(* IEC 61131-3 sources: teller/JD_Teller_LC2_V11/Class/Box_Editer, 1 file *)

(* ---- Box_Editer.st ---- *)
(*!
<Class
	Name               = "Box_Editer"
	Revision           = "1.7"
	RealtimeTask       = "false"
	CyclicTask         = "false"
	BackgroundTask     = "false"
	Sigmatek           = "false"
	OSInterface        = "false"
	HighPriority       = "false"
	Automatic          = "false"
	UpdateMode         = "Prescan"
	SharedCommandTable = "true"
	Objectsize         = "(750,1860)">
	<Channels>
		<Server Name="ClassSvr" Visualized="false" Initialize="false" WriteProtected="true" Retentive="false"/>
		<Server Name="Parameter_Ok" Visualized="true" Initialize="false" WriteProtected="true" Retentive="false" Comment="Visu&#13;&#10;&#13;&#10;Als een doos berekend wordt dan wordt &#13;&#10;er gecontroleerd of de parameters kloppen&#13;&#10;&#13;&#10;Bij&#13;&#10;0: Fout&#13;&#10;1: Goed&#13;&#10;&#13;&#10;De servers T_Status, en verder geven de foute waarden per parameter aan&#13;&#10;"/>
		<Server Name="Presets_MinMax" Visualized="true" Initialize="false" WriteProtected="false" Retentive="false"/>
		<Server Name="ResetValues" Visualized="true" Initialize="false" WriteProtected="false" Retentive="false"/>
		<Server Name="s_BoxMogelijkopMachine" Visualized="true" Initialize="false" WriteProtected="false" Retentive="false" Comment="Is deze doos te draaien op de machine?&#13;&#10;&#13;&#10;0: nee&#13;&#10;1: ja&#13;&#10;"/>
		<Server Name="s_BoxType" Visualized="true" Initialize="false" WriteProtected="false" Retentive="SRam"/>
		<Server Name="s_Calc_Box" Visualized="true" Initialize="false" WriteProtected="false" Retentive="false"/>
		<Server Name="s_Doosnaam" Visualized="true" Initialize="false" WriteProtected="true" Retentive="false"/>
		<Server Name="s_MaxLength" Visualized="true" Initialize="false" WriteProtected="false" Retentive="false"/>
		<Server Name="s_MaxWidth" Visualized="true" Initialize="false" WriteProtected="false" Retentive="false"/>
		<Server Name="s_Offset" Visualized="true" Initialize="false" WriteProtected="false" Retentive="false"/>
		<Server Name="s_Offset_Max" Visualized="true" Initialize="false" WriteProtected="false" Retentive="false"/>
		<Server Name="s_Offset_Min" Visualized="true" Initialize="false" WriteProtected="false" Retentive="false"/>
		<Server Name="s_Refresh_Values" Visualized="false" Initialize="false" WriteProtected="false" Retentive="false"/>
		<Server Name="s_T" Visualized="true" Initialize="false" WriteProtected="false" Retentive="false"/>
		<Server Name="s_T_Max" Visualized="true" Initialize="false" WriteProtected="false" Retentive="false"/>
		<Server Name="s_T_Min" Visualized="true" Initialize="false" WriteProtected="false" Retentive="false"/>
		<Server Name="s_U" Visualized="true" Initialize="false" WriteProtected="false" Retentive="false"/>
		<Server Name="s_U_Max" Visualized="true" Initialize="false" WriteProtected="false" Retentive="false"/>
		<Server Name="s_U_Min" Visualized="true" Initialize="false" WriteProtected="false" Retentive="false"/>
		<Server Name="s_V" Visualized="true" Initialize="false" WriteProtected="false" Retentive="false"/>
		<Server Name="s_V_Max" Visualized="true" Initialize="false" WriteProtected="false" Retentive="false"/>
		<Server Name="s_V_Min" Visualized="true" Initialize="false" WriteProtected="false" Retentive="false"/>
		<Server Name="s_W" Visualized="true" Initialize="false" WriteProtected="false" Retentive="false"/>
		<Server Name="s_W_Max" Visualized="true" Initialize="false" WriteProtected="false" Retentive="false"/>
		<Server Name="s_W_Min" Visualized="true" Initialize="false" WriteProtected="false" Retentive="false"/>
		<Server Name="s_X" Visualized="true" Initialize="false" WriteProtected="false" Retentive="false"/>
		<Server Name="s_X_Max" Visualized="true" Initialize="false" WriteProtected="false" Retentive="false"/>
		<Server Name="s_X_Min" Visualized="true" Initialize="false" WriteProtected="false" Retentive="false"/>
		<Server Name="s_Y" Visualized="true" Initialize="false" WriteProtected="false" Retentive="false"/>
		<Server Name="s_Y_Max" Visualized="true" Initialize="false" WriteProtected="false" Retentive="false"/>
		<Server Name="s_Y_Min" Visualized="true" Initialize="false" WriteProtected="false" Retentive="false"/>
		<Server Name="s_Z" Visualized="true" Initialize="false" WriteProtected="false" Retentive="false"/>
		<Server Name="s_Z_Max" Visualized="true" Initialize="false" WriteProtected="false" Retentive="false"/>
		<Server Name="s_Z_Min" Visualized="true" Initialize="false" WriteProtected="false" Retentive="false"/>
		<Server Name="T_Status" Visualized="true" Initialize="false" WriteProtected="true" Retentive="false"/>
		<Server Name="U_Status" Visualized="true" Initialize="false" WriteProtected="true" Retentive="false"/>
		<Server Name="V_Status" Visualized="true" Initialize="false" WriteProtected="true" Retentive="false"/>
		<Server Name="W_Status" Visualized="true" Initialize="false" WriteProtected="true" Retentive="false"/>
		<Server Name="X_Status" Visualized="true" Initialize="false" WriteProtected="true" Retentive="false"/>
		<Server Name="Y_Status" Visualized="true" Initialize="false" WriteProtected="true" Retentive="false"/>
		<Server Name="Z_Status" Visualized="true" Initialize="false" WriteProtected="true" Retentive="false"/>
		<Client Name="c_DoosData" Required="true" Internal="false"/>
		<Client Name="c_Mask_Out" Required="true" Internal="false"/>
		<Client Name="c_Refresh_Preview" Required="true" Internal="false"/>
		<Client Name="c_Refresh_Values01" Required="false" Internal="false"/>
		<Client Name="c_Refresh_Values02" Required="false" Internal="false"/>
		<Client Name="c_Refresh_Values03" Required="false" Internal="false"/>
		<Client Name="c_Refresh_Values04" Required="false" Internal="false"/>
		<Client Name="c_Refresh_Values05" Required="false" Internal="false"/>
		<Client Name="c_Refresh_Values06" Required="false" Internal="false"/>
		<Client Name="c_Refresh_Values07" Required="false" Internal="false"/>
		<Client Name="c_Refresh_Values08" Required="false" Internal="false"/>
		<Client Name="c_Refresh_Values09" Required="false" Internal="false"/>
		<Client Name="c_Refresh_Values10" Required="false" Internal="false"/>
		<Client Name="c_Refresh_Values11" Required="false" Internal="false"/>
		<Client Name="c_Refresh_Values12" Required="false" Internal="false"/>
		<Client Name="c_Refresh_Values13" Required="true" Internal="false"/>
		<Client Name="c_Refresh_Values14" Required="true" Internal="false"/>
		<Client Name="c_UpdatePrefold" Required="true" Internal="false"/>
		<Client Name="c_WriteCalc" Required="false" Internal="false"/>
	</Channels>
	<RevDoku>
		<Owner Company="JD" Author="J van Diggelen"/>
		<Dokumentation Revision="1.7" Date="2014-04-22" Author="J van Diggelen" Company="JD" Description="Doos14 toegevoegd"/>
		<Dokumentation Revision="1.6" Date="2014-01-27" Author="J van Diggelen" Company="JD" Description="Mask wordt uitgestuurd"/>
		<Dokumentation Revision="1.5" Date="2013-09-21" Author="J van Diggelen" Company="JD" Description="Warning parameter never used verwijderd"/>
		<Dokumentation Revision="1.4" Date="2013-08-21" Author="J van Diggelen" Company="JD" Description="client aanpassing ivm prefold knop"/>
		<Dokumentation Revision="1.3" Date="2012-08-28" Author="J van Diggelen" Company="JD" Description="-Doostype 13 toegevoegd"/>
		<Dokumentation Revision="1.2" Date="2012-08-02" Author="J van Diggelen" Company="JD" Description="-Extra server aangemaakt ResetValues Dit om bij nieuwe doos de doosdata op 0 te zetten"/>
		<Dokumentation Revision="1.1" Date="2012-01-30" Author="J van Diggelen" Company="JD" Description="-Bij boxtype 0 wordt er een Maximale length van 2000 in de init ingevoerd. &#13;&#10;Dit om bij de lijm een spoor in te kunnen geven."/>
		<Dokumentation Revision="1.0" Date="2011-12-06" Author="J van Diggelen" Company="JD" Description="-Boxeditor is uitgebreid zodat er per type doos de service instellingen kan worden ingegeven"/>
	</RevDoku>
</Class>
*)
Box_Editer : CLASS
  //Servers:
	ClassSvr 	: SvrChCmd_DINT;
	s_Doosnaam 	: SvrCh_tDoosnaam;
	s_BoxType 	: SvrCh_DINT;
	s_BoxMogelijkopMachine 	: SvrCh_DINT;
	Presets_MinMax 	: SvrCh_tModel;
	s_T 	: SvrCh_DINT;
	s_U 	: SvrCh_DINT;
	s_V 	: SvrCh_DINT;
	s_W 	: SvrCh_DINT;
	s_X 	: SvrCh_DINT;
	s_Y 	: SvrCh_DINT;
	s_Z 	: SvrCh_DINT;
	s_Offset 	: SvrCh_DINT;
	s_MaxLength 	: SvrCh_DINT;
	s_MaxWidth 	: SvrCh_DINT;
	s_T_Max 	: SvrCh_DINT;
	s_T_Min 	: SvrCh_DINT;
	s_U_Max 	: SvrCh_DINT;
	s_U_Min 	: SvrCh_DINT;
	s_V_Max 	: SvrCh_DINT;
	s_V_Min 	: SvrCh_DINT;
	s_W_Max 	: SvrCh_DINT;
	s_W_Min 	: SvrCh_DINT;
	s_X_Max 	: SvrCh_DINT;
	s_X_Min 	: SvrCh_DINT;
	s_Y_Max 	: SvrCh_DINT;
	s_Y_Min 	: SvrCh_DINT;
	s_Z_Max 	: SvrCh_DINT;
	s_Z_Min 	: SvrCh_DINT;
	s_Offset_Max 	: SvrCh_DINT;
	s_Offset_Min 	: SvrCh_DINT;
	s_Refresh_Values 	: SvrCh_DINT;
	s_Calc_Box 	: SvrCh_DINT;
	Parameter_Ok 	: SvrCh_DINT;
	T_Status 	: SvrCh_DINT;
	U_Status 	: SvrCh_DINT;
	V_Status 	: SvrCh_DINT;
	W_Status 	: SvrCh_DINT;
	X_Status 	: SvrCh_DINT;
	Y_Status 	: SvrCh_DINT;
	Z_Status 	: SvrCh_DINT;
	ResetValues 	: SvrCh_DINT;
  //Clients:
	c_DoosData 	: CltChCmd_RAMex;
	c_Refresh_Preview 	: CltCh_DINT;
	c_Refresh_Values01 	: CltCh_DINT;
	c_Refresh_Values02 	: CltCh_DINT;
	c_Refresh_Values03 	: CltCh_DINT;
	c_Refresh_Values04 	: CltCh_DINT;
	c_Refresh_Values05 	: CltCh_DINT;
	c_Refresh_Values06 	: CltCh_DINT;
	c_Refresh_Values07 	: CltCh_DINT;
	c_Refresh_Values08 	: CltCh_DINT;
	c_Refresh_Values09 	: CltCh_DINT;
	c_Refresh_Values10 	: CltCh_DINT;
	c_Refresh_Values11 	: CltCh_DINT;
	c_Refresh_Values12 	: CltCh_DINT;
	c_Refresh_Values13 	: CltCh_DINT;
	c_Refresh_Values14 	: CltCh_DINT;
	c_WriteCalc 	: CltCh_DINT;
	c_UpdatePrefold 	: CltCh_DINT;
	c_Mask_Out 	: CltCh_DINT;
  //Variables:
		DoosData 	: ^tDoosParameters;
		i 	: DINT;
  //Functions:

	FUNCTION VIRTUAL GLOBAL Init;

	FUNCTION VIRTUAL GLOBAL Background
		VAR_INPUT
			EAX 	: UDINT;
		END_VAR
		VAR_OUTPUT
			state (EAX) 	: UDINT;
		END_VAR;

	FUNCTION Refesh;

	FUNCTION VIRTUAL GLOBAL s_BoxType::Write
		VAR_INPUT
			input (EAX) 	: DINT;
		END_VAR
		VAR_OUTPUT
			result (EAX) 	: DINT;
		END_VAR;

	FUNCTION VIRTUAL GLOBAL s_BoxMogelijkopMachine::Write
		VAR_INPUT
			input (EAX) 	: DINT;
		END_VAR
		VAR_OUTPUT
			result (EAX) 	: DINT;
		END_VAR;

	FUNCTION VIRTUAL GLOBAL Presets_MinMax::Write
		VAR_INPUT
			input (EAX) 	: tModel;
		END_VAR
		VAR_OUTPUT
			result (EAX) 	: tModel;
		END_VAR;

	FUNCTION VIRTUAL GLOBAL s_T::Write
		VAR_INPUT
			input (EAX) 	: DINT;
		END_VAR
		VAR_OUTPUT
			result (EAX) 	: DINT;
		END_VAR;

	FUNCTION VIRTUAL GLOBAL s_U::Write
		VAR_INPUT
			input (EAX) 	: DINT;
		END_VAR
		VAR_OUTPUT
			result (EAX) 	: DINT;
		END_VAR;

	FUNCTION VIRTUAL GLOBAL s_V::Write
		VAR_INPUT
			input (EAX) 	: DINT;
		END_VAR
		VAR_OUTPUT
			result (EAX) 	: DINT;
		END_VAR;

	FUNCTION VIRTUAL GLOBAL s_W::Write
		VAR_INPUT
			input (EAX) 	: DINT;
		END_VAR
		VAR_OUTPUT
			result (EAX) 	: DINT;
		END_VAR;

	FUNCTION VIRTUAL GLOBAL s_X::Write
		VAR_INPUT
			input (EAX) 	: DINT;
		END_VAR
		VAR_OUTPUT
			result (EAX) 	: DINT;
		END_VAR;

	FUNCTION VIRTUAL GLOBAL s_Y::Write
		VAR_INPUT
			input (EAX) 	: DINT;
		END_VAR
		VAR_OUTPUT
			result (EAX) 	: DINT;
		END_VAR;

	FUNCTION VIRTUAL GLOBAL s_Z::Write
		VAR_INPUT
			input (EAX) 	: DINT;
		END_VAR
		VAR_OUTPUT
			result (EAX) 	: DINT;
		END_VAR;

	FUNCTION VIRTUAL GLOBAL s_Offset::Write
		VAR_INPUT
			input (EAX) 	: DINT;
		END_VAR
		VAR_OUTPUT
			result (EAX) 	: DINT;
		END_VAR;

	FUNCTION VIRTUAL GLOBAL s_MaxLength::Write
		VAR_INPUT
			input (EAX) 	: DINT;
		END_VAR
		VAR_OUTPUT
			result (EAX) 	: DINT;
		END_VAR;

	FUNCTION VIRTUAL GLOBAL s_MaxWidth::Write
		VAR_INPUT
			input (EAX) 	: DINT;
		END_VAR
		VAR_OUTPUT
			result (EAX) 	: DINT;
		END_VAR;

	FUNCTION VIRTUAL GLOBAL s_T_Max::Write
		VAR_INPUT
			input (EAX) 	: DINT;
		END_VAR
		VAR_OUTPUT
			result (EAX) 	: DINT;
		END_VAR;

	FUNCTION VIRTUAL GLOBAL s_T_Min::Write
		VAR_INPUT
			input (EAX) 	: DINT;
		END_VAR
		VAR_OUTPUT
			result (EAX) 	: DINT;
		END_VAR;

	FUNCTION VIRTUAL GLOBAL s_U_Max::Write
		VAR_INPUT
			input (EAX) 	: DINT;
		END_VAR
		VAR_OUTPUT
			result (EAX) 	: DINT;
		END_VAR;

	FUNCTION VIRTUAL GLOBAL s_U_Min::Write
		VAR_INPUT
			input (EAX) 	: DINT;
		END_VAR
		VAR_OUTPUT
			result (EAX) 	: DINT;
		END_VAR;

	FUNCTION VIRTUAL GLOBAL s_V_Max::Write
		VAR_INPUT
			input (EAX) 	: DINT;
		END_VAR
		VAR_OUTPUT
			result (EAX) 	: DINT;
		END_VAR;

	FUNCTION VIRTUAL GLOBAL s_V_Min::Write
		VAR_INPUT
			input (EAX) 	: DINT;
		END_VAR
		VAR_OUTPUT
			result (EAX) 	: DINT;
		END_VAR;

	FUNCTION VIRTUAL GLOBAL s_W_Max::Write
		VAR_INPUT
			input (EAX) 	: DINT;
		END_VAR
		VAR_OUTPUT
			result (EAX) 	: DINT;
		END_VAR;

	FUNCTION VIRTUAL GLOBAL s_W_Min::Write
		VAR_INPUT
			input (EAX) 	: DINT;
		END_VAR
		VAR_OUTPUT
			result (EAX) 	: DINT;
		END_VAR;

	FUNCTION VIRTUAL GLOBAL s_X_Max::Write
		VAR_INPUT
			input (EAX) 	: DINT;
		END_VAR
		VAR_OUTPUT
			result (EAX) 	: DINT;
		END_VAR;

	FUNCTION VIRTUAL GLOBAL s_X_Min::Write
		VAR_INPUT
			input (EAX) 	: DINT;
		END_VAR
		VAR_OUTPUT
			result (EAX) 	: DINT;
		END_VAR;

	FUNCTION VIRTUAL GLOBAL s_Y_Max::Write
		VAR_INPUT
			input (EAX) 	: DINT;
		END_VAR
		VAR_OUTPUT
			result (EAX) 	: DINT;
		END_VAR;

	FUNCTION VIRTUAL GLOBAL s_Y_Min::Write
		VAR_INPUT
			input (EAX) 	: DINT;
		END_VAR
		VAR_OUTPUT
			result (EAX) 	: DINT;
		END_VAR;

	FUNCTION VIRTUAL GLOBAL s_Z_Max::Write
		VAR_INPUT
			input (EAX) 	: DINT;
		END_VAR
		VAR_OUTPUT
			result (EAX) 	: DINT;
		END_VAR;

	FUNCTION VIRTUAL GLOBAL s_Z_Min::Write
		VAR_INPUT
			input (EAX) 	: DINT;
		END_VAR
		VAR_OUTPUT
			result (EAX) 	: DINT;
		END_VAR;

	FUNCTION VIRTUAL GLOBAL s_Offset_Max::Write
		VAR_INPUT
			input (EAX) 	: DINT;
		END_VAR
		VAR_OUTPUT
			result (EAX) 	: DINT;
		END_VAR;

	FUNCTION VIRTUAL GLOBAL s_Offset_Min::Write
		VAR_INPUT
			input (EAX) 	: DINT;
		END_VAR
		VAR_OUTPUT
			result (EAX) 	: DINT;
		END_VAR;

	FUNCTION VIRTUAL GLOBAL s_Refresh_Values::Write
		VAR_INPUT
			input (EAX) 	: DINT;
		END_VAR
		VAR_OUTPUT
			result (EAX) 	: DINT;
		END_VAR;

	FUNCTION VIRTUAL GLOBAL s_Calc_Box::Write
		VAR_INPUT
			input (EAX) 	: DINT;
		END_VAR
		VAR_OUTPUT
			result (EAX) 	: DINT;
		END_VAR;

	FUNCTION VIRTUAL GLOBAL ResetValues::Write
		VAR_INPUT
			input (EAX) 	: DINT;
		END_VAR
		VAR_OUTPUT
			result (EAX) 	: DINT;
		END_VAR;
  //Tables:
	FUNCTION @STD
		VAR_OUTPUT
			ret_code	: CONFSTATES;
		END_VAR;
	FUNCTION GLOBAL TAB @CT_;
END_CLASS;

#pragma usingLtd RAMex

//Er is in de pointer variabele doosdata een array structuur gemaakt om bij elk type doos de minimale en maximale
//waardes in een service scherm te veranderen.

FUNCTION VIRTUAL GLOBAL Box_Editer::Init

  if c_DoosData.GetSize() <> sizeof(tDoosParameters) then
     c_DoosData.SetSize(udSize:=sizeof(tDoosParameters));
  end_if;

  if _FirstScan = 1 then

  DoosData := (c_DoosData.GetDataPtr())$^tDoosParameters;
//     s_BoxType := 0;
//     DoosData^.Doostype :=0;
//     s_BoxType.Write(0);

  s_BoxType.Write(input:=s_BoxType);

  s_T:=DoosData^.T;
  c_Mask_Out.Write(input:=s_T);
  s_U:=DoosData^.U;
  s_V:=DoosData^.V;
  s_W:=DoosData^.W;
  s_X:=DoosData^.X;
  s_Y:=DoosData^.Y;
  s_Z:=DoosData^.Z;
  s_Offset:=DoosData^.Offset;

  if s_MaxLength <= 0 then
     s_MaxLength := (2000);
  end_if;

  end_if;

END_FUNCTION

FUNCTION VIRTUAL GLOBAL Box_Editer::Background
	VAR_INPUT
		EAX 	: UDINT;
	END_VAR
	VAR_OUTPUT
		state (EAX) 	: UDINT;
	END_VAR

	state := READY;

END_FUNCTION

FUNCTION VIRTUAL GLOBAL Box_Editer::s_BoxType::Write
	VAR_INPUT
		input (EAX) 	: DINT;
	END_VAR
	VAR_OUTPUT
		result (EAX) 	: DINT;
	END_VAR

	s_BoxType := input;

  // doostype moet tussen 0 en 14 liggen
  if    s_BoxType <0 then
        s_BoxType :=0;
  elsif s_BoxType >14 then
        s_BoxType :=14;
  end_if;

 	result := s_BoxType;

  //Nummerieke doostype
  DoosData^.Doostype := s_BoxType;
  c_UpdatePrefold.Write(input:=1);
  //Doostype
  if     s_BoxType = 0 then
         s_Doosnaam := No_box;
  elsif  s_BoxType = 1 then
         s_Doosnaam := Langsnaad;
  elsif  s_BoxType = 2 then
         s_Doosnaam := Driepunt;
  elsif  s_BoxType = 3 then
         s_Doosnaam := Driepunt_Vakverdeling;
  elsif  s_BoxType = 4 then
         s_Doosnaam := Vierpunt_Infold;
  elsif  s_BoxType = 5 then
         s_Doosnaam := Vierpunt_Outfold;
  elsif  s_BoxType = 6 then
         s_Doosnaam := Vierpunt_Deksel;
  elsif  s_BoxType = 7 then
         s_Doosnaam := Vierpunt_Dubbele_Wand;
  elsif  s_BoxType = 8 then
         s_Doosnaam := Zespunt_In_In;
  elsif  s_BoxType = 9 then
         s_Doosnaam := Zespunt_In_Out;
  elsif  s_BoxType = 10 then
         s_Doosnaam := Zespunt_In_In_Gespiegeld;
  elsif  s_BoxType = 11 then
         s_Doosnaam := Driepunt_Gespiegeld;
  elsif  s_BoxType = 12 then
         s_Doosnaam := Driepunt;
  elsif  s_BoxType = 13 then
         s_Doosnaam := Langsnaad2;
  elsif  s_BoxType = 14 then
         s_Doosnaam := Driepunt2;
  end_if;

  //Serverwaardes schrijven met variabelen voor type doos
  if s_BoxType <> 0 then
    s_MaxLength := DoosData^.MinMax[s_BoxType].Max_Invoer_Lengte;
    s_MaxWidth  := DoosData^.MinMax[s_BoxType].Max_Invoer_Breedte;
    s_BoxMogelijkopMachine := DoosData^.MinMax[s_BoxType].BoxMogelijk;
    s_T_Max     := DoosData^.MinMax[s_BoxType].T_Max;
    s_T_Min     := DoosData^.MinMax[s_BoxType].T_Min;
    s_U_Max     := DoosData^.MinMax[s_BoxType].U_Max;
    s_U_Min     := DoosData^.MinMax[s_BoxType].U_Min;
    s_V_Min     := DoosData^.MinMax[s_BoxType].V_Min;
    s_V_Max     := DoosData^.MinMax[s_BoxType].V_Max;
    s_W_Max     := DoosData^.MinMax[s_BoxType].W_Max;
    s_W_Min     := DoosData^.MinMax[s_BoxType].W_Min;
    s_X_Max     := DoosData^.MinMax[s_BoxType].X_Max;
    s_X_Min     := DoosData^.MinMax[s_BoxType].X_Min;
    s_Y_Max     := DoosData^.MinMax[s_BoxType].Y_Max;
    s_Y_Min     := DoosData^.MinMax[s_BoxType].Y_Min;
    s_Z_Max     := DoosData^.MinMax[s_BoxType].Z_Max;
    s_Z_Min     := DoosData^.MinMax[s_BoxType].Z_Min;
    s_Offset_Max:= DoosData^.MinMax[s_BoxType].Offset_Max;
    s_Offset_Min:= DoosData^.MinMax[s_BoxType].Offset_Min;
  end_if;

END_FUNCTION

FUNCTION VIRTUAL GLOBAL Box_Editer::s_BoxMogelijkopMachine::Write
	VAR_INPUT
		input (EAX) 	: DINT;
	END_VAR
	VAR_OUTPUT
		result (EAX) 	: DINT;
	END_VAR

	s_BoxMogelijkopMachine := input;
  DoosData^.MinMax[s_BoxType].BoxMogelijk := to_bool(s_BoxMogelijkopMachine);

  if      s_BoxType = 1 then
          c_Refresh_Values01.Write(input:=1);
  elsif   s_BoxType = 2 then
          c_Refresh_Values02.Write(input:=1);
  elsif   s_BoxType = 3 then
          c_Refresh_Values03.Write(input:=1);
  elsif   s_BoxType = 4 then
          c_Refresh_Values04.Write(input:=1);
  elsif   s_BoxType = 5 then
          c_Refresh_Values05.Write(input:=1);
  elsif   s_BoxType = 6 then
          c_Refresh_Values06.Write(input:=1);
  elsif   s_BoxType = 7 then
          c_Refresh_Values07.Write(input:=1);
  elsif   s_BoxType = 8 then
          c_Refresh_Values08.Write(input:=1);
  elsif   s_BoxType = 9 then
          c_Refresh_Values09.Write(input:=1);
  elsif   s_BoxType = 10 then
          c_Refresh_Values10.Write(input:=1);
  elsif   s_BoxType = 11 then
          c_Refresh_Values11.Write(input:=1);
  elsif   s_BoxType = 12 then
          c_Refresh_Values12.Write(input:=1);
  elsif   s_BoxType = 13 then
          c_Refresh_Values13.Write(input:=1);
  elsif   s_BoxType = 14 then
          c_Refresh_Values14.Write(input:=1);
  end_if;

 	result := s_BoxMogelijkopMachine;

END_FUNCTION

FUNCTION VIRTUAL GLOBAL Box_Editer::s_T::Write
	VAR_INPUT
		input (EAX) 	: DINT;
	END_VAR
	VAR_OUTPUT
		result (EAX) 	: DINT;
	END_VAR

	s_T := input;
  DoosData^.T := s_T;
  c_Mask_Out.Write(input:=s_T);
 	result := s_T;

  c_Refresh_Preview.Write(input:=1);

END_FUNCTION

FUNCTION VIRTUAL GLOBAL Box_Editer::s_U::Write
	VAR_INPUT
		input (EAX) 	: DINT;
	END_VAR
	VAR_OUTPUT
		result (EAX) 	: DINT;
	END_VAR

	s_U := input;
  DoosData^.U := s_U;
 	result := s_U;

  c_Refresh_Preview.Write(input:=1);

END_FUNCTION

FUNCTION VIRTUAL GLOBAL Box_Editer::s_V::Write
	VAR_INPUT
		input (EAX) 	: DINT;
	END_VAR
	VAR_OUTPUT
		result (EAX) 	: DINT;
	END_VAR

	s_V := input;
 	DoosData^.V := s_V;
  result := s_V;

  c_Refresh_Preview.Write(input:=1);

END_FUNCTION

FUNCTION VIRTUAL GLOBAL Box_Editer::s_W::Write
	VAR_INPUT
		input (EAX) 	: DINT;
	END_VAR
	VAR_OUTPUT
		result (EAX) 	: DINT;
	END_VAR

	s_W := input;
  DoosData^.W := s_W;
 	result := s_W;

  c_Refresh_Preview.Write(input:=1);

END_FUNCTION

FUNCTION VIRTUAL GLOBAL Box_Editer::s_X::Write
	VAR_INPUT
		input (EAX) 	: DINT;
	END_VAR
	VAR_OUTPUT
		result (EAX) 	: DINT;
	END_VAR

	s_X := input;
  DoosData^.X := s_X;
  result := s_X;

  c_Refresh_Preview.Write(input:=1);

END_FUNCTION

FUNCTION VIRTUAL GLOBAL Box_Editer::s_Y::Write
	VAR_INPUT
		input (EAX) 	: DINT;
	END_VAR
	VAR_OUTPUT
		result (EAX) 	: DINT;
	END_VAR

	s_Y := input;
  DoosData^.Y := s_Y;
 	result := s_Y;

  c_Refresh_Preview.Write(input:=1);

END_FUNCTION

FUNCTION VIRTUAL GLOBAL Box_Editer::s_Z::Write
	VAR_INPUT
		input (EAX) 	: DINT;
	END_VAR
	VAR_OUTPUT
		result (EAX) 	: DINT;
	END_VAR

	s_Z := input;
  DoosData^.Z := s_Z;
 	result := s_Z;

  c_Refresh_Preview.Write(input:=1);

END_FUNCTION

FUNCTION VIRTUAL GLOBAL Box_Editer::s_Offset::Write
	VAR_INPUT
		input (EAX) 	: DINT;
	END_VAR
	VAR_OUTPUT
		result (EAX) 	: DINT;
	END_VAR

	s_Offset := input;
  DoosData^.Offset := s_Offset;
 	result := s_Offset;

  c_Refresh_Preview.Write(input:=1);

END_FUNCTION

FUNCTION VIRTUAL GLOBAL Box_Editer::s_MaxLength::Write
	VAR_INPUT
		input (EAX) 	: DINT;
	END_VAR
	VAR_OUTPUT
		result (EAX) 	: DINT;
	END_VAR

	s_MaxLength := input;
  DoosData^.MinMax[s_BoxType].Max_Invoer_Lengte := s_MaxLength;
  Refesh(); //Refresh de MinMax classes door met de client te schrijven
 	result := s_MaxLength;

END_FUNCTION

FUNCTION VIRTUAL GLOBAL Box_Editer::s_MaxWidth::Write
	VAR_INPUT
		input (EAX) 	: DINT;
	END_VAR
	VAR_OUTPUT
		result (EAX) 	: DINT;
	END_VAR

	s_MaxWidth := input;
  DoosData^.MinMax[s_BoxType].Max_Invoer_Breedte := s_MaxWidth;
  Refesh(); //Refresh de MinMax classes door met de client te schrijven
 	result := s_MaxWidth;

END_FUNCTION

FUNCTION VIRTUAL GLOBAL Box_Editer::s_T_Max::Write
	VAR_INPUT
		input (EAX) 	: DINT;
	END_VAR
	VAR_OUTPUT
		result (EAX) 	: DINT;
	END_VAR

	s_T_Max := input;
  DoosData^.MinMax[s_BoxType].T_Max:= s_T_Max;
  Refesh(); //Refresh de MinMax classes door met de client te schrijven
 	result := s_T_Max;

END_FUNCTION

FUNCTION VIRTUAL GLOBAL Box_Editer::s_T_Min::Write
	VAR_INPUT
		input (EAX) 	: DINT;
	END_VAR
	VAR_OUTPUT
		result (EAX) 	: DINT;
	END_VAR

	s_T_Min := input;
  DoosData^.MinMax[s_BoxType].T_Min:= s_T_Min;
  Refesh(); //Refresh de MinMax classes door met de client te schrijven
 	result := s_T_Min;

END_FUNCTION

FUNCTION VIRTUAL GLOBAL Box_Editer::s_U_Max::Write
	VAR_INPUT
		input (EAX) 	: DINT;
	END_VAR
	VAR_OUTPUT
		result (EAX) 	: DINT;
	END_VAR

	s_U_Max := input;
  DoosData^.MinMax[s_BoxType].U_Max:=s_U_Max;
  Refesh(); //Refresh de MinMax classes door met de client te schrijven
 	result := s_U_Max;

END_FUNCTION

FUNCTION VIRTUAL GLOBAL Box_Editer::s_U_Min::Write
	VAR_INPUT
		input (EAX) 	: DINT;
	END_VAR
	VAR_OUTPUT
		result (EAX) 	: DINT;
	END_VAR

	s_U_Min := input;
  DoosData^.MinMax[s_BoxType].U_Min:= s_U_Min;
  Refesh(); //Refresh de MinMax classes door met de client te schrijven
 	result := s_U_Min;

END_FUNCTION

FUNCTION VIRTUAL GLOBAL Box_Editer::s_V_Max::Write
	VAR_INPUT
		input (EAX) 	: DINT;
	END_VAR
	VAR_OUTPUT
		result (EAX) 	: DINT;
	END_VAR

	s_V_Max := input;
  DoosData^.MinMax[s_BoxType].V_Max:=s_V_Max;
  Refesh(); //Refresh de MinMax classes door met de client te schrijven
 	result := s_V_Max;

END_FUNCTION

FUNCTION VIRTUAL GLOBAL Box_Editer::s_V_Min::Write
	VAR_INPUT
		input (EAX) 	: DINT;
	END_VAR
	VAR_OUTPUT
		result (EAX) 	: DINT;
	END_VAR

	s_V_Min := input;
  DoosData^.MinMax[s_BoxType].V_Min:=s_V_Min;
  Refesh(); //Refresh de MinMax classes door met de client te schrijven
 	result := s_V_Min;

END_FUNCTION

FUNCTION VIRTUAL GLOBAL Box_Editer::s_W_Max::Write
	VAR_INPUT
		input (EAX) 	: DINT;
	END_VAR
	VAR_OUTPUT
		result (EAX) 	: DINT;
	END_VAR

	s_W_Max := input;
  DoosData^.MinMax[s_BoxType].W_Max:=s_W_Max;
  Refesh(); //Refresh de MinMax classes door met de client te schrijven
 	result := s_W_Max;

END_FUNCTION

FUNCTION VIRTUAL GLOBAL Box_Editer::s_W_Min::Write
	VAR_INPUT
		input (EAX) 	: DINT;
	END_VAR
	VAR_OUTPUT
		result (EAX) 	: DINT;
	END_VAR

	s_W_Min := input;
  DoosData^.MinMax[s_BoxType].W_Min:=s_W_Min;
  Refesh(); //Refresh de MinMax classes door met de client te schrijven
 	result := s_W_Min;

END_FUNCTION

FUNCTION VIRTUAL GLOBAL Box_Editer::s_X_Max::Write
	VAR_INPUT
		input (EAX) 	: DINT;
	END_VAR
	VAR_OUTPUT
		result (EAX) 	: DINT;
	END_VAR

	s_X_Max := input;
  DoosData^.MinMax[s_BoxType].X_Max:=s_X_Max;
  Refesh(); //Refresh de MinMax classes door met de client te schrijven
 	result := s_X_Max;

END_FUNCTION

FUNCTION VIRTUAL GLOBAL Box_Editer::s_X_Min::Write
	VAR_INPUT
		input (EAX) 	: DINT;
	END_VAR
	VAR_OUTPUT
		result (EAX) 	: DINT;
	END_VAR

	s_X_Min := input;
  DoosData^.MinMax[s_BoxType].X_Min:=s_X_Min;
  Refesh(); //Refresh de MinMax classes door met de client te schrijven
 	result := s_X_Min;

END_FUNCTION

FUNCTION VIRTUAL GLOBAL Box_Editer::s_Y_Max::Write
	VAR_INPUT
		input (EAX) 	: DINT;
	END_VAR
	VAR_OUTPUT
		result (EAX) 	: DINT;
	END_VAR

	s_Y_Max := input;
  DoosData^.MinMax[s_BoxType].Y_Max:=s_Y_Max;
  Refesh(); //Refresh de MinMax classes door met de client te schrijven
 	result := s_Y_Max;

END_FUNCTION

FUNCTION VIRTUAL GLOBAL Box_Editer::s_Y_Min::Write
	VAR_INPUT
		input (EAX) 	: DINT;
	END_VAR
	VAR_OUTPUT
		result (EAX) 	: DINT;
	END_VAR

	s_Y_Min := input;
  DoosData^.MinMax[s_BoxType].Y_Min:= s_Y_Min;
  Refesh(); //Refresh de MinMax classes door met de client te schrijven
 	result := s_Y_Min;

END_FUNCTION

FUNCTION VIRTUAL GLOBAL Box_Editer::s_Z_Max::Write
	VAR_INPUT
		input (EAX) 	: DINT;
	END_VAR
	VAR_OUTPUT
		result (EAX) 	: DINT;
	END_VAR

	s_Z_Max := input;
  DoosData^.MinMax[s_BoxType].Z_Max:= s_Z_Max;
  Refesh(); //Refresh de MinMax classes door met de client te schrijven
 	result := s_Z_Max;

END_FUNCTION

FUNCTION VIRTUAL GLOBAL Box_Editer::s_Z_Min::Write
	VAR_INPUT
		input (EAX) 	: DINT;
	END_VAR
	VAR_OUTPUT
		result (EAX) 	: DINT;
	END_VAR

	s_Z_Min := input;
  DoosData^.MinMax[s_BoxType].Z_Min:= s_Z_Min;
  Refesh(); //Refresh de MinMax classes door met de client te schrijven
 	result := s_Z_Min;

END_FUNCTION

FUNCTION VIRTUAL GLOBAL Box_Editer::s_Offset_Max::Write
	VAR_INPUT
		input (EAX) 	: DINT;
	END_VAR
	VAR_OUTPUT
		result (EAX) 	: DINT;
	END_VAR

	s_Offset_Max := input;
  DoosData^.MinMax[s_BoxType].Offset_Max:= s_Offset_Max;
  Refesh(); //Refresh de MinMax classes door met de client te schrijven
 	result := s_Offset_Max;

END_FUNCTION

FUNCTION VIRTUAL GLOBAL Box_Editer::s_Offset_Min::Write
	VAR_INPUT
		input (EAX) 	: DINT;
	END_VAR
	VAR_OUTPUT
		result (EAX) 	: DINT;
	END_VAR

	s_Offset_Min := input;
  DoosData^.MinMax[s_BoxType].Offset_Min:= s_Offset_Min;
  Refesh(); //Refresh de MinMax classes door met de client te schrijven
 	result := s_Offset_Min;

END_FUNCTION

FUNCTION Box_Editer::Refesh

  if      s_BoxType = 1 then
          c_Refresh_Values01.Write(input:=1);
  elsif   s_BoxType = 2 then
          c_Refresh_Values02.Write(input:=1);
  elsif   s_BoxType = 3 then
          c_Refresh_Values03.Write(input:=1);
  elsif   s_BoxType = 4 then
          c_Refresh_Values04.Write(input:=1);
  elsif   s_BoxType = 5 then
          c_Refresh_Values05.Write(input:=1);
  elsif   s_BoxType = 6 then
          c_Refresh_Values06.Write(input:=1);
  elsif   s_BoxType = 7 then
          c_Refresh_Values07.Write(input:=1);
  elsif   s_BoxType = 8 then
          c_Refresh_Values08.Write(input:=1);
  elsif   s_BoxType = 9 then
          c_Refresh_Values09.Write(input:=1);
  elsif   s_BoxType = 10 then
          c_Refresh_Values10.Write(input:=1);
  elsif   s_BoxType = 11 then
          c_Refresh_Values11.Write(input:=1);
  elsif   s_BoxType = 12 then
          c_Refresh_Values12.Write(input:=1);
  elsif   s_BoxType = 13 then
          c_Refresh_Values13.Write(input:=1);
  elsif   s_BoxType = 14 then
          c_Refresh_Values14.Write(input:=1);
  end_if;

END_FUNCTION

FUNCTION VIRTUAL GLOBAL Box_Editer::s_Refresh_Values::Write

	VAR_INPUT
		input (EAX) 	: DINT;
	END_VAR
	VAR_OUTPUT
		result (EAX) 	: DINT;
	END_VAR

	s_Refresh_Values := input;
  s_Refresh_Values := 0;
  s_BoxType.Write(s_BoxType);
 	result := s_Refresh_Values;

END_FUNCTION

FUNCTION VIRTUAL GLOBAL Box_Editer::s_Calc_Box::Write
	VAR_INPUT
		input (EAX) 	: DINT;
	END_VAR
	VAR_OUTPUT
		result (EAX) 	: DINT;
	END_VAR

	s_Calc_Box := input;
  s_Calc_Box := 0;

  Parameter_Ok := 0;
  T_Status := 1;
  U_Status := 1;
  V_Status := 1;
  W_Status := 1;
  X_Status := 1;
  Y_Status := 1;
  Z_Status := 1;

    //langsnaad
  if    Doosdata^.Doostype = 1 then

        if    Doosdata^.X >= Doosdata^.W then
              X_Status := 0;
              W_Status := 0;
        end_if;
        if    Doosdata^.Y >= Doosdata^.W then
              Y_Status := 0;
              W_Status := 0;
        end_if;

        if    (2*Doosdata^.X + 2*Doosdata^.Y) >= Doosdata^.W then
              X_Status := 0;
              Y_Status := 0;
              W_Status := 0;
        end_if;

        if    (2*Doosdata^.U) >= Doosdata^.T then
              T_Status := 0;
              U_Status := 0;
        end_if;

        if    Doosdata^.Z > 150 then
              Z_Status := 0;
        end_if;

        if    T_Status = 1 &
              U_Status = 1 &
              V_Status = 1 &
              W_Status = 1 &
              X_Status = 1 &
              Y_Status = 1 &
              Z_Status = 1 then
              Parameter_Ok := 1;
        end_if;

  //3-punt
  elsif Doosdata^.Doostype = 2 then

        if    Doosdata^.X >= Doosdata^.W then
              X_Status := 0;
              W_Status := 0;
        end_if;
        if    Doosdata^.Y >= Doosdata^.W then
              Y_Status := 0;
              W_Status := 0;
        end_if;

        if    (2*Doosdata^.X + 2*Doosdata^.Y) >= Doosdata^.W then
              X_Status := 0;
              Y_Status := 0;
              W_Status := 0;
        end_if;

        if    (2*Doosdata^.U) >= Doosdata^.T then
              T_Status := 0;
              U_Status := 0;
        end_if;

        if    (2*Doosdata^.V) >= Doosdata^.T then
              V_Status := 0;
              U_Status := 0;
        end_if;

        if    Doosdata^.Z > 150 then
              Z_Status := 0;
        end_if;

        if    T_Status = 1 &
              U_Status = 1 &
              V_Status = 1 &
              W_Status = 1 &
              X_Status = 1 &
              Y_Status = 1 &
              Z_Status = 1 then
              Parameter_Ok := 1;
        end_if;

  //3-punt vakverdeling
  elsif Doosdata^.Doostype = 3 then

        if    Doosdata^.X >= Doosdata^.W then
              X_Status := 0;
              W_Status := 0;
        end_if;
        if    Doosdata^.Y >= Doosdata^.W then
              Y_Status := 0;
              W_Status := 0;
        end_if;

        if    (2*Doosdata^.X + 2*Doosdata^.Y) >= Doosdata^.W then
              X_Status := 0;
              Y_Status := 0;
              W_Status := 0;
        end_if;

        if    (2*Doosdata^.U) >= Doosdata^.T then
              T_Status := 0;
              U_Status := 0;
        end_if;

        if    (2*Doosdata^.V) >= Doosdata^.T then
              V_Status := 0;
              U_Status := 0;
        end_if;

        if    Doosdata^.Z > 150 then
              Z_Status := 0;
        end_if;

        if    T_Status = 1 &
              U_Status = 1 &
              V_Status = 1 &
              W_Status = 1 &
              X_Status = 1 &
              Y_Status = 1 &
              Z_Status = 1 then
              Parameter_Ok := 1;
        end_if;

  //4-punt infold
  elsif Doosdata^.Doostype = 4 then

        if    (2*Doosdata^.U) >= Doosdata^.T then
              T_Status := 0;
              U_Status := 0;
        end_if;

        if    (2*Doosdata^.V) >= Doosdata^.T then
              V_Status := 0;
              U_Status := 0;
        end_if;

        if    Doosdata^.Z > 150 then
              Z_Status := 0;
        end_if;

        if    T_Status = 1 &
              U_Status = 1 &
              V_Status = 1 &
              W_Status = 1 &
              X_Status = 1 &
              Y_Status = 1 &
              Z_Status = 1 then
              Parameter_Ok := 1;
        end_if;

  //4-punt outfold
  elsif Doosdata^.Doostype = 5 then

        if    (2*Doosdata^.U) >= Doosdata^.T then
              T_Status := 0;
              U_Status := 0;
        end_if;

        if    Doosdata^.Z > 150 then
              Z_Status := 0;
        end_if;

        if    T_Status = 1 &
              U_Status = 1 &
              V_Status = 1 &
              W_Status = 1 &
              X_Status = 1 &
              Y_Status = 1 &
              Z_Status = 1 then
              Parameter_Ok := 1;
        end_if;

  //4-punt met deksel
  elsif Doosdata^.Doostype = 6 then

        if    Doosdata^.X >= Doosdata^.W then
              X_Status := 0;
              W_Status := 0;
        end_if;
        if    Doosdata^.Y >= Doosdata^.W then
              Y_Status := 0;
              W_Status := 0;
        end_if;

        if    (2*Doosdata^.X + 2*Doosdata^.Y) >= Doosdata^.W then
              X_Status := 0;
              Y_Status := 0;
              W_Status := 0;
        end_if;

        if    (2*Doosdata^.U) >= Doosdata^.T then
              T_Status := 0;
              U_Status := 0;
        end_if;

        if    (2*Doosdata^.V) >= Doosdata^.T then
              V_Status := 0;
              U_Status := 0;
        end_if;

        if    Doosdata^.Z > 150 then
              Z_Status := 0;
        end_if;

        if    T_Status = 1 &
              U_Status = 1 &
              V_Status = 1 &
              W_Status = 1 &
              X_Status = 1 &
              Y_Status = 1 &
              Z_Status = 1 then
              Parameter_Ok := 1;
        end_if;

  //4-punt dubbele wand
  elsif Doosdata^.Doostype = 7 then

        if    Doosdata^.X >= Doosdata^.W then
              X_Status := 0;
              W_Status := 0;
        end_if;
        if    Doosdata^.Y >= Doosdata^.W then
              Y_Status := 0;
              W_Status := 0;
        end_if;

        if    (4*Doosdata^.X + Doosdata^.Y) > Doosdata^.W then
              X_Status := 0;
              Y_Status := 0;
              W_Status := 0;
        end_if;

        if    (2*Doosdata^.U) >= Doosdata^.T then
              T_Status := 0;
              U_Status := 0;
        end_if;

        if    (2*Doosdata^.V) >= Doosdata^.T then
              V_Status := 0;
              U_Status := 0;
        end_if;

        if    Doosdata^.Z > 150 then
              Z_Status := 0;
        end_if;

        if    T_Status = 1 &
              U_Status = 1 &
              V_Status = 1 &
              W_Status = 1 &
              X_Status = 1 &
              Y_Status = 1 &
              Z_Status = 1 then
              Parameter_Ok := 1;
        end_if;

  //6-punt in/in
  elsif Doosdata^.Doostype = 8 then

        if    Doosdata^.X >= Doosdata^.W then
              X_Status := 0;
              W_Status := 0;
        end_if;

        if    Doosdata^.Y >= Doosdata^.W then
              Y_Status := 0;
              W_Status := 0;
        end_if;

        if    (3*Doosdata^.X + 2*Doosdata^.Y) > Doosdata^.W then
              X_Status := 0;
              Y_Status := 0;
              W_Status := 0;
        end_if;

        if    (2*Doosdata^.U) >= Doosdata^.T then
              T_Status := 0;
              U_Status := 0;
        end_if;

        if    (2*Doosdata^.V) >= Doosdata^.T then
              V_Status := 0;
              U_Status := 0;
        end_if;

        if    Doosdata^.Z > 150 then
              Z_Status := 0;
        end_if;

        if    T_Status = 1 &
              U_Status = 1 &
              V_Status = 1 &
              W_Status = 1 &
              X_Status = 1 &
              Y_Status = 1 &
              Z_Status = 1 then
              Parameter_Ok := 1;
        end_if;

  //6-punt in/out
  elsif Doosdata^.Doostype = 9 then

        if    Doosdata^.X >= Doosdata^.W then
              X_Status := 0;
              W_Status := 0;
        end_if;

        if    Doosdata^.Y >= Doosdata^.W then
              Y_Status := 0;
              W_Status := 0;
        end_if;

        if    (3*Doosdata^.X + 2*Doosdata^.Y) > Doosdata^.W then
              X_Status := 0;
              Y_Status := 0;
              W_Status := 0;
        end_if;

        if    (2*Doosdata^.U) >= Doosdata^.T then
              T_Status := 0;
              U_Status := 0;
        end_if;

        if    (2*Doosdata^.V) >= Doosdata^.T then
              V_Status := 0;
              U_Status := 0;
        end_if;

        if    Doosdata^.Z > 150 then
              Z_Status := 0;
        end_if;

        if    T_Status = 1 &
              U_Status = 1 &
              V_Status = 1 &
              W_Status = 1 &
              X_Status = 1 &
              Y_Status = 1 &
              Z_Status = 1 then
              Parameter_Ok := 1;
        end_if;

  //6-punt in/in
  elsif Doosdata^.Doostype = 10 then

        if    Doosdata^.X >= Doosdata^.W then
              X_Status := 0;
              W_Status := 0;
        end_if;

        if    Doosdata^.Y >= Doosdata^.W then
              Y_Status := 0;
              W_Status := 0;
        end_if;

        if    (3*Doosdata^.X + 2*Doosdata^.Y) > Doosdata^.W then
              X_Status := 0;
              Y_Status := 0;
              W_Status := 0;
        end_if;

        if    (2*Doosdata^.U) >= Doosdata^.T then
              T_Status := 0;
              U_Status := 0;
        end_if;

        if    (2*Doosdata^.V) >= Doosdata^.T then
              V_Status := 0;
              U_Status := 0;
        end_if;

        if    Doosdata^.Z > 150 then
              Z_Status := 0;
        end_if;

        if    T_Status = 1 &
              U_Status = 1 &
              V_Status = 1 &
              W_Status = 1 &
              X_Status = 1 &
              Y_Status = 1 &
              Z_Status = 1 then
              Parameter_Ok := 1;
        end_if;

  //3-punt (gespiegeld)
  elsif Doosdata^.Doostype = 11 then

        if    Doosdata^.X >= Doosdata^.W then
              X_Status := 0;
              W_Status := 0;
        end_if;
        if    Doosdata^.Y >= Doosdata^.W then
              Y_Status := 0;
              W_Status := 0;
        end_if;

        if    (2*Doosdata^.X + 2*Doosdata^.Y) >= Doosdata^.W then
              X_Status := 0;
              Y_Status := 0;
              W_Status := 0;
        end_if;

        if    (2*Doosdata^.U) >= Doosdata^.T then
              T_Status := 0;
              U_Status := 0;
        end_if;

        if    (2*Doosdata^.V) >= Doosdata^.T then
              V_Status := 0;
              U_Status := 0;
        end_if;

        if    Doosdata^.Z > 150 then
              Z_Status := 0;
        end_if;

        if    T_Status = 1 &
              U_Status = 1 &
              V_Status = 1 &
              W_Status = 1 &
              X_Status = 1 &
              Y_Status = 1 &
              Z_Status = 1 then
              Parameter_Ok := 1;
        end_if;

  //3-punt (Storaenzo Jonkoping)
  elsif Doosdata^.Doostype = 12 then

        if    Doosdata^.X >= Doosdata^.W then
              X_Status := 0;
              W_Status := 0;
        end_if;
        if    Doosdata^.Y >= Doosdata^.W then
              Y_Status := 0;
              W_Status := 0;
        end_if;

        if    (2*Doosdata^.X + 2*Doosdata^.Y) >= Doosdata^.W then
              X_Status := 0;
              Y_Status := 0;
              W_Status := 0;
        end_if;

        if    (2*Doosdata^.U) >= Doosdata^.T then
              T_Status := 0;
              U_Status := 0;
        end_if;

        if    (2*Doosdata^.V) >= Doosdata^.T then
              V_Status := 0;
              U_Status := 0;
        end_if;

        if    Doosdata^.Z > 150 then
              Z_Status := 0;
        end_if;

        if    T_Status = 1 &
              U_Status = 1 &
              V_Status = 1 &
              W_Status = 1 &
              X_Status = 1 &
              Y_Status = 1 &
              Z_Status = 1 then
              Parameter_Ok := 1;
        end_if;

    //langsnaad2
  elsif Doosdata^.Doostype = 13 then

        if    Doosdata^.X >= Doosdata^.W then
              X_Status := 0;
              W_Status := 0;
        end_if;
        if    Doosdata^.Y >= Doosdata^.W then
              Y_Status := 0;
              W_Status := 0;
        end_if;

        if    (2*Doosdata^.X + 2*Doosdata^.Y) >= Doosdata^.W then
              X_Status := 0;
              Y_Status := 0;
              W_Status := 0;
        end_if;

        if    (2*Doosdata^.U) >= Doosdata^.T then
              T_Status := 0;
              U_Status := 0;
        end_if;

        if    (2*Doosdata^.V) >= Doosdata^.T then
              T_Status := 0;
              V_Status := 0;
        end_if;

        if    Doosdata^.Z > 150 then
              Z_Status := 0;
        end_if;

        if    T_Status = 1 &
              U_Status = 1 &
              V_Status = 1 &
              W_Status = 1 &
              X_Status = 1 &
              Y_Status = 1 &
              Z_Status = 1 then
              Parameter_Ok := 1;
        end_if;

  //3-punt2 (SK Soest)
  elsif Doosdata^.Doostype = 14 then

        if    Doosdata^.X >= Doosdata^.W then
              X_Status := 0;
              W_Status := 0;
        end_if;
        if    Doosdata^.Y >= Doosdata^.W then
              Y_Status := 0;
              W_Status := 0;
        end_if;

        if    (2*Doosdata^.X + 2*Doosdata^.Y) >= Doosdata^.W then
              X_Status := 0;
              Y_Status := 0;
              W_Status := 0;
        end_if;

        if    (2*Doosdata^.U) >= Doosdata^.T then
              T_Status := 0;
              U_Status := 0;
        end_if;

        if    (2*Doosdata^.V) >= Doosdata^.T then
              V_Status := 0;
              U_Status := 0;
        end_if;

        if    Doosdata^.Z > 150 then
              Z_Status := 0;
        end_if;

        if    T_Status = 1 &
              U_Status = 1 &
              V_Status = 1 &
              W_Status = 1 &
              X_Status = 1 &
              Y_Status = 1 &
              Z_Status = 1 then
              Parameter_Ok := 1;
        end_if;

  end_if;

  if  Parameter_Ok = 1 then
      c_Mask_Out.Write(input:=Doosdata^.T);
      c_WriteCalc.Write(1);
  end_if;

 	result := s_Calc_Box;

END_FUNCTION

FUNCTION VIRTUAL GLOBAL Box_Editer::Presets_MinMax::Write
	VAR_INPUT
		input (EAX) 	: tModel;
	END_VAR
	VAR_OUTPUT
		result (EAX) 	: tModel;
	END_VAR

	Presets_MinMax := input;

  if    Presets_MinMax =  m1250 then

        for i:= 1 to 14 do

            DoosData^.MinMax[i].Max_Invoer_Lengte  := 2000;
            DoosData^.MinMax[i].Max_Invoer_Breedte := 1250;

              //langsnaad 1250
            if    i = 1 then

                  DoosData^.MinMax[i].T_Max := 2000;
                  DoosData^.MinMax[i].T_Min := 70;
                  DoosData^.MinMax[i].U_Max := 300;
                  DoosData^.MinMax[i].U_Min := 30;
                  DoosData^.MinMax[i].V_Max := 0;
                  DoosData^.MinMax[i].V_Min := 0;
                  DoosData^.MinMax[i].W_Max := 1250;
                  DoosData^.MinMax[i].W_Min := 270;
                  DoosData^.MinMax[i].X_Max := 450;
                  DoosData^.MinMax[i].X_Min := 30;
                  DoosData^.MinMax[i].Y_Max := 450;
                  DoosData^.MinMax[i].Y_Min := 70;
                  DoosData^.MinMax[i].Z_Max := 3000;
                  DoosData^.MinMax[i].Z_Min := 0;
                  DoosData^.MinMax[i].Offset_Max := 625;
                  DoosData^.MinMax[i].Offset_Min := 0;

            //3-punt 1250
            elsif i = 2 then

                  DoosData^.MinMax[i].T_Max := 2000;
                  DoosData^.MinMax[i].T_Min := 70;
                  DoosData^.MinMax[i].U_Max := 200;
                  DoosData^.MinMax[i].U_Min := 30;
                  DoosData^.MinMax[i].V_Max := 200;
                  DoosData^.MinMax[i].V_Min := 30;
                  DoosData^.MinMax[i].W_Max := 1250;
                  DoosData^.MinMax[i].W_Min := 270;
                  DoosData^.MinMax[i].X_Max := 450;
                  DoosData^.MinMax[i].X_Min := 40;
                  DoosData^.MinMax[i].Y_Max := 450;
                  DoosData^.MinMax[i].Y_Min := 70;
                  DoosData^.MinMax[i].Z_Max := 3000;
                  DoosData^.MinMax[i].Z_Min := 0;
                  DoosData^.MinMax[i].Offset_Max := 625;
                  DoosData^.MinMax[i].Offset_Min := 0;

            //3-punt vakverdeling 1250
            elsif i = 3 then

                  DoosData^.MinMax[i].T_Max := 2000;
                  DoosData^.MinMax[i].T_Min := 160;
                  DoosData^.MinMax[i].U_Max := 300;
                  DoosData^.MinMax[i].U_Min := 30;
                  DoosData^.MinMax[i].V_Max := 300;
                  DoosData^.MinMax[i].V_Min := 30;
                  DoosData^.MinMax[i].W_Max := 1100;
                  DoosData^.MinMax[i].W_Min := 400;
                  DoosData^.MinMax[i].X_Max := 500;
                  DoosData^.MinMax[i].X_Min := 110;
                  DoosData^.MinMax[i].Y_Max := 500;
                  DoosData^.MinMax[i].Y_Min := 90;
                  DoosData^.MinMax[i].Z_Max := 3000;
                  DoosData^.MinMax[i].Z_Min := 0;
                  DoosData^.MinMax[i].Offset_Max := 625;
                  DoosData^.MinMax[i].Offset_Min := 0;

            //4-punt infold 1250
            elsif i = 4 then

                  DoosData^.MinMax[i].T_Max := 2000;
                  DoosData^.MinMax[i].T_Min := 80;
                  DoosData^.MinMax[i].U_Max := 300;
                  DoosData^.MinMax[i].U_Min := 30;
                  DoosData^.MinMax[i].V_Max := 300;
                  DoosData^.MinMax[i].V_Min := 30;
                  DoosData^.MinMax[i].W_Max := 0;
                  DoosData^.MinMax[i].W_Min := 0;
                  DoosData^.MinMax[i].X_Max := 150;
                  DoosData^.MinMax[i].X_Min := 30;
                  DoosData^.MinMax[i].Y_Max := 680;
                  DoosData^.MinMax[i].Y_Min := 130;
                  DoosData^.MinMax[i].Z_Max := 3000;
                  DoosData^.MinMax[i].Z_Min := 0;
                  DoosData^.MinMax[i].Offset_Max := 625;
                  DoosData^.MinMax[i].Offset_Min := 0;

            //4-punt outfold 1250
            elsif i = 5 then

                  DoosData^.MinMax[i].T_Max := 2000;
                  DoosData^.MinMax[i].T_Min := 80;
                  DoosData^.MinMax[i].U_Max := 300;
                  DoosData^.MinMax[i].U_Min := 30;
                  DoosData^.MinMax[i].V_Max := 300;
                  DoosData^.MinMax[i].V_Min := 30;
                  DoosData^.MinMax[i].W_Max := 0;
                  DoosData^.MinMax[i].W_Min := 0;
                  DoosData^.MinMax[i].X_Max := 300;
                  DoosData^.MinMax[i].X_Min := 30;
                  DoosData^.MinMax[i].Y_Max := 680;
                  DoosData^.MinMax[i].Y_Min := 130;
                  DoosData^.MinMax[i].Z_Max := 3000;
                  DoosData^.MinMax[i].Z_Min := 0;
                  DoosData^.MinMax[i].Offset_Max := 625;
                  DoosData^.MinMax[i].Offset_Min := 0;

            //4-punt met deksel 1250
            elsif i = 6 then

                  DoosData^.MinMax[i].T_Max := 2000;
                  DoosData^.MinMax[i].T_Min := 80;
                  DoosData^.MinMax[i].U_Max := 300;
                  DoosData^.MinMax[i].U_Min := 30;
                  DoosData^.MinMax[i].V_Max := 300;
                  DoosData^.MinMax[i].V_Min := 30;
                  DoosData^.MinMax[i].W_Max := 1100;
                  DoosData^.MinMax[i].W_Min := 0;
                  DoosData^.MinMax[i].X_Max := 150;
                  DoosData^.MinMax[i].X_Min := 30;
                  DoosData^.MinMax[i].Y_Max := 680;
                  DoosData^.MinMax[i].Y_Min := 130;
                  DoosData^.MinMax[i].Z_Max := 3000;
                  DoosData^.MinMax[i].Z_Min := 0;
                  DoosData^.MinMax[i].Offset_Max := 625;
                  DoosData^.MinMax[i].Offset_Min := 0;

            //4-punt dubbele wand 1250
            elsif i = 7 then

                  DoosData^.MinMax[i].T_Max := 2000;
                  DoosData^.MinMax[i].T_Min := 80;
                  DoosData^.MinMax[i].U_Max := 300;
                  DoosData^.MinMax[i].U_Min := 30;
                  DoosData^.MinMax[i].V_Max := 300;
                  DoosData^.MinMax[i].V_Min := 30;
                  DoosData^.MinMax[i].W_Max := 1100;
                  DoosData^.MinMax[i].W_Min := 0;
                  DoosData^.MinMax[i].X_Max := 150;
                  DoosData^.MinMax[i].X_Min := 30;
                  DoosData^.MinMax[i].Y_Max := 680;
                  DoosData^.MinMax[i].Y_Min := 130;
                  DoosData^.MinMax[i].Z_Max := 3000;
                  DoosData^.MinMax[i].Z_Min := 0;
                  DoosData^.MinMax[i].Offset_Max := 625;
                  DoosData^.MinMax[i].Offset_Min := 0;

            //6-punt in/in 1250
            elsif i = 8 then

                  DoosData^.MinMax[i].T_Max := 2000;
                  DoosData^.MinMax[i].T_Min := 80;
                  DoosData^.MinMax[i].U_Max := 300;
                  DoosData^.MinMax[i].U_Min := 30;
                  DoosData^.MinMax[i].V_Max := 300;
                  DoosData^.MinMax[i].V_Min := 30;
                  DoosData^.MinMax[i].W_Max := 1100;
                  DoosData^.MinMax[i].W_Min := 0;
                  DoosData^.MinMax[i].X_Max := 150;
                  DoosData^.MinMax[i].X_Min := 30;
                  DoosData^.MinMax[i].Y_Max := 680;
                  DoosData^.MinMax[i].Y_Min := 130;
                  DoosData^.MinMax[i].Z_Max := 3000;
                  DoosData^.MinMax[i].Z_Min := 0;
                  DoosData^.MinMax[i].Offset_Max := 625;
                  DoosData^.MinMax[i].Offset_Min := 0;

            //6-punt in/out 1250
            elsif i = 9 then

                  DoosData^.MinMax[i].T_Max := 2000;
                  DoosData^.MinMax[i].T_Min := 80;
                  DoosData^.MinMax[i].U_Max := 300;
                  DoosData^.MinMax[i].U_Min := 30;
                  DoosData^.MinMax[i].V_Max := 300;
                  DoosData^.MinMax[i].V_Min := 30;
                  DoosData^.MinMax[i].W_Max := 1100;
                  DoosData^.MinMax[i].W_Min := 0;
                  DoosData^.MinMax[i].X_Max := 150;
                  DoosData^.MinMax[i].X_Min := 30;
                  DoosData^.MinMax[i].Y_Max := 680;
                  DoosData^.MinMax[i].Y_Min := 130;
                  DoosData^.MinMax[i].Z_Max := 3000;
                  DoosData^.MinMax[i].Z_Min := 0;
                  DoosData^.MinMax[i].Offset_Max := 625;
                  DoosData^.MinMax[i].Offset_Min := 0;

            //6-punt in/in 1250
            elsif i = 10 then

                  DoosData^.MinMax[i].T_Max := 2000;
                  DoosData^.MinMax[i].T_Min := 80;
                  DoosData^.MinMax[i].U_Max := 300;
                  DoosData^.MinMax[i].U_Min := 30;
                  DoosData^.MinMax[i].V_Max := 300;
                  DoosData^.MinMax[i].V_Min := 30;
                  DoosData^.MinMax[i].W_Max := 1100;
                  DoosData^.MinMax[i].W_Min := 0;
                  DoosData^.MinMax[i].X_Max := 150;
                  DoosData^.MinMax[i].X_Min := 30;
                  DoosData^.MinMax[i].Y_Max := 680;
                  DoosData^.MinMax[i].Y_Min := 130;
                  DoosData^.MinMax[i].Z_Max := 3000;
                  DoosData^.MinMax[i].Z_Min := 0;
                  DoosData^.MinMax[i].Offset_Max := 625;
                  DoosData^.MinMax[i].Offset_Min := 0;

            //3-punt (gespiegeld) 1250
            elsif i = 11 then

                  DoosData^.MinMax[i].T_Max := 2000;
                  DoosData^.MinMax[i].T_Min := 70;
                  DoosData^.MinMax[i].U_Max := 200;
                  DoosData^.MinMax[i].U_Min := 30;
                  DoosData^.MinMax[i].V_Max := 200;
                  DoosData^.MinMax[i].V_Min := 30;
                  DoosData^.MinMax[i].W_Max := 1250;
                  DoosData^.MinMax[i].W_Min := 270;
                  DoosData^.MinMax[i].X_Max := 450;
                  DoosData^.MinMax[i].X_Min := 40;
                  DoosData^.MinMax[i].Y_Max := 450;
                  DoosData^.MinMax[i].Y_Min := 70;
                  DoosData^.MinMax[i].Z_Max := 3000;
                  DoosData^.MinMax[i].Z_Min := 0;
                  DoosData^.MinMax[i].Offset_Max := 625;
                  DoosData^.MinMax[i].Offset_Min := 0;

            //3-punt (Storaenzo Jonkoping) 1250
            elsif i = 12 then

                  DoosData^.MinMax[i].T_Max := 2000;
                  DoosData^.MinMax[i].T_Min := 70;
                  DoosData^.MinMax[i].U_Max := 200;
                  DoosData^.MinMax[i].U_Min := 30;
                  DoosData^.MinMax[i].V_Max := 200;
                  DoosData^.MinMax[i].V_Min := 30;
                  DoosData^.MinMax[i].W_Max := 1250;
                  DoosData^.MinMax[i].W_Min := 270;
                  DoosData^.MinMax[i].X_Max := 450;
                  DoosData^.MinMax[i].X_Min := 40;
                  DoosData^.MinMax[i].Y_Max := 450;
                  DoosData^.MinMax[i].Y_Min := 70;
                  DoosData^.MinMax[i].Z_Max := 3000;
                  DoosData^.MinMax[i].Z_Min := 0;
                  DoosData^.MinMax[i].Offset_Max := 625;
                  DoosData^.MinMax[i].Offset_Min := 0;

            //langsnaad2 1250
            elsif i = 13 then

                  DoosData^.MinMax[i].T_Max := 2000;
                  DoosData^.MinMax[i].T_Min := 70;
                  DoosData^.MinMax[i].U_Max := 300;
                  DoosData^.MinMax[i].U_Min := 30;
                  DoosData^.MinMax[i].V_Max := 300;
                  DoosData^.MinMax[i].V_Min := 30;
                  DoosData^.MinMax[i].W_Max := 1250;
                  DoosData^.MinMax[i].W_Min := 270;
                  DoosData^.MinMax[i].X_Max := 450;
                  DoosData^.MinMax[i].X_Min := 30;
                  DoosData^.MinMax[i].Y_Max := 450;
                  DoosData^.MinMax[i].Y_Min := 70;
                  DoosData^.MinMax[i].Z_Max := 3000;
                  DoosData^.MinMax[i].Z_Min := 0;
                  DoosData^.MinMax[i].Offset_Max := 625;
                  DoosData^.MinMax[i].Offset_Min := 0;

            //3-punt2 1250
            elsif i = 14 then

                  DoosData^.MinMax[i].T_Max := 2000;
                  DoosData^.MinMax[i].T_Min := 70;
                  DoosData^.MinMax[i].U_Max := 200;
                  DoosData^.MinMax[i].U_Min := 30;
                  DoosData^.MinMax[i].V_Max := 200;
                  DoosData^.MinMax[i].V_Min := 30;
                  DoosData^.MinMax[i].W_Max := 1250;
                  DoosData^.MinMax[i].W_Min := 270;
                  DoosData^.MinMax[i].X_Max := 450;
                  DoosData^.MinMax[i].X_Min := 40;
                  DoosData^.MinMax[i].Y_Max := 450;
                  DoosData^.MinMax[i].Y_Min := 70;
                  DoosData^.MinMax[i].Z_Max := 3000;
                  DoosData^.MinMax[i].Z_Min := 0;
                  DoosData^.MinMax[i].Offset_Max := 625;
                  DoosData^.MinMax[i].Offset_Min := 0;

            end_if;
        end_for;
  end_if;

  if    Presets_MinMax =  m1450 then

        for i:= 1 to 14 do

            DoosData^.MinMax[i].Max_Invoer_Lengte  := 2000;
            DoosData^.MinMax[i].Max_Invoer_Breedte := 1450;

              //langsnaad 1450
            if    i = 1 then

                  DoosData^.MinMax[i].T_Max := 2000;
                  DoosData^.MinMax[i].T_Min := 100;
                  DoosData^.MinMax[i].U_Max := 300;
                  DoosData^.MinMax[i].U_Min := 40;
                  DoosData^.MinMax[i].V_Max := 0;
                  DoosData^.MinMax[i].V_Min := 0;
                  DoosData^.MinMax[i].W_Max := 1450;
                  DoosData^.MinMax[i].W_Min := 320;
                  DoosData^.MinMax[i].X_Max := 525;
                  DoosData^.MinMax[i].X_Min := 40;
                  DoosData^.MinMax[i].Y_Max := 525;
                  DoosData^.MinMax[i].Y_Min := 75;
                  DoosData^.MinMax[i].Z_Max := 3000;
                  DoosData^.MinMax[i].Z_Min := 0;
                  DoosData^.MinMax[i].Offset_Max := 725;
                  DoosData^.MinMax[i].Offset_Min := 0;

            //3-punt 1450
            elsif i = 2 then

                  DoosData^.MinMax[i].T_Max := 2000;
                  DoosData^.MinMax[i].T_Min := 100;
                  DoosData^.MinMax[i].U_Max := 250;
                  DoosData^.MinMax[i].U_Min := 40;
                  DoosData^.MinMax[i].V_Max := 250;
                  DoosData^.MinMax[i].V_Min := 40;
                  DoosData^.MinMax[i].W_Max := 1450;
                  DoosData^.MinMax[i].W_Min := 320;
                  DoosData^.MinMax[i].X_Max := 525;
                  DoosData^.MinMax[i].X_Min := 50;
                  DoosData^.MinMax[i].Y_Max := 525;
                  DoosData^.MinMax[i].Y_Min := 75;
                  DoosData^.MinMax[i].Z_Max := 3000;
                  DoosData^.MinMax[i].Z_Min := 0;
                  DoosData^.MinMax[i].Offset_Max := 725;
                  DoosData^.MinMax[i].Offset_Min := 0;

            //3-punt vakverdeling 1450
            elsif i = 3 then

                  DoosData^.MinMax[i].T_Max := 2000;
                  DoosData^.MinMax[i].T_Min := 200;
                  DoosData^.MinMax[i].U_Max := 300;
                  DoosData^.MinMax[i].U_Min := 30;
                  DoosData^.MinMax[i].V_Max := 300;
                  DoosData^.MinMax[i].V_Min := 30;
                  DoosData^.MinMax[i].W_Max := 1300;
                  DoosData^.MinMax[i].W_Min := 400;
                  DoosData^.MinMax[i].X_Max := 500;
                  DoosData^.MinMax[i].X_Min := 110;
                  DoosData^.MinMax[i].Y_Max := 500;
                  DoosData^.MinMax[i].Y_Min := 90;
                  DoosData^.MinMax[i].Z_Max := 3000;
                  DoosData^.MinMax[i].Z_Min := 0;
                  DoosData^.MinMax[i].Offset_Max := 725;
                  DoosData^.MinMax[i].Offset_Min := 0;

            //4-punt infold 1450
            elsif i = 4 then

                  DoosData^.MinMax[i].T_Max := 2000;
                  DoosData^.MinMax[i].T_Min := 100;
                  DoosData^.MinMax[i].U_Max := 300;
                  DoosData^.MinMax[i].U_Min := 30;
                  DoosData^.MinMax[i].V_Max := 300;
                  DoosData^.MinMax[i].V_Min := 30;
                  DoosData^.MinMax[i].W_Max := 0;
                  DoosData^.MinMax[i].W_Min := 0;
                  DoosData^.MinMax[i].X_Max := 300;
                  DoosData^.MinMax[i].X_Min := 30;
                  DoosData^.MinMax[i].Y_Max := 980;
                  DoosData^.MinMax[i].Y_Min := 155;
                  DoosData^.MinMax[i].Z_Max := 3000;
                  DoosData^.MinMax[i].Z_Min := 0;
                  DoosData^.MinMax[i].Offset_Max := 725;
                  DoosData^.MinMax[i].Offset_Min := 0;

            //4-punt outfold 1450
            elsif i = 5 then

                  DoosData^.MinMax[i].T_Max := 2000;
                  DoosData^.MinMax[i].T_Min := 100;
                  DoosData^.MinMax[i].U_Max := 300;
                  DoosData^.MinMax[i].U_Min := 30;
                  DoosData^.MinMax[i].V_Max := 300;
                  DoosData^.MinMax[i].V_Min := 30;
                  DoosData^.MinMax[i].W_Max := 0;
                  DoosData^.MinMax[i].W_Min := 0;
                  DoosData^.MinMax[i].X_Max := 300;
                  DoosData^.MinMax[i].X_Min := 30;
                  DoosData^.MinMax[i].Y_Max := 980;
                  DoosData^.MinMax[i].Y_Min := 155;
                  DoosData^.MinMax[i].Z_Max := 3000;
                  DoosData^.MinMax[i].Z_Min := 0;
                  DoosData^.MinMax[i].Offset_Max := 725;
                  DoosData^.MinMax[i].Offset_Min := 0;

            //4-punt met deksel 1450
            elsif i = 6 then

                  DoosData^.MinMax[i].T_Max := 2000;
                  DoosData^.MinMax[i].T_Min := 100;
                  DoosData^.MinMax[i].U_Max := 300;
                  DoosData^.MinMax[i].U_Min := 30;
                  DoosData^.MinMax[i].V_Max := 300;
                  DoosData^.MinMax[i].V_Min := 30;
                  DoosData^.MinMax[i].W_Max := 1280;
                  DoosData^.MinMax[i].W_Min := 0;
                  DoosData^.MinMax[i].X_Max := 300;
                  DoosData^.MinMax[i].X_Min := 30;
                  DoosData^.MinMax[i].Y_Max := 980;
                  DoosData^.MinMax[i].Y_Min := 155;
                  DoosData^.MinMax[i].Z_Max := 3000;
                  DoosData^.MinMax[i].Z_Min := 0;
                  DoosData^.MinMax[i].Offset_Max := 725;
                  DoosData^.MinMax[i].Offset_Min := 0;

            //4-punt dubbele wand 1450
            elsif i = 7 then

                  DoosData^.MinMax[i].T_Max := 2000;
                  DoosData^.MinMax[i].T_Min := 100;
                  DoosData^.MinMax[i].U_Max := 300;
                  DoosData^.MinMax[i].U_Min := 30;
                  DoosData^.MinMax[i].V_Max := 300;
                  DoosData^.MinMax[i].V_Min := 30;
                  DoosData^.MinMax[i].W_Max := 1280;
                  DoosData^.MinMax[i].W_Min := 0;
                  DoosData^.MinMax[i].X_Max := 300;
                  DoosData^.MinMax[i].X_Min := 30;
                  DoosData^.MinMax[i].Y_Max := 980;
                  DoosData^.MinMax[i].Y_Min := 155;
                  DoosData^.MinMax[i].Z_Max := 3000;
                  DoosData^.MinMax[i].Z_Min := 0;
                  DoosData^.MinMax[i].Offset_Max := 725;
                  DoosData^.MinMax[i].Offset_Min := 0;

            //6-punt in/in 1450
            elsif i = 8 then

                  DoosData^.MinMax[i].T_Max := 2000;
                  DoosData^.MinMax[i].T_Min := 100;
                  DoosData^.MinMax[i].U_Max := 300;
                  DoosData^.MinMax[i].U_Min := 30;
                  DoosData^.MinMax[i].V_Max := 300;
                  DoosData^.MinMax[i].V_Min := 30;
                  DoosData^.MinMax[i].W_Max := 1280;
                  DoosData^.MinMax[i].W_Min := 0;
                  DoosData^.MinMax[i].X_Max := 300;
                  DoosData^.MinMax[i].X_Min := 30;
                  DoosData^.MinMax[i].Y_Max := 980;
                  DoosData^.MinMax[i].Y_Min := 155;
                  DoosData^.MinMax[i].Z_Max := 3000;
                  DoosData^.MinMax[i].Z_Min := 0;
                  DoosData^.MinMax[i].Offset_Max := 725;
                  DoosData^.MinMax[i].Offset_Min := 0;

            //6-punt in/out 1450
            elsif i = 9 then

                  DoosData^.MinMax[i].T_Max := 2000;
                  DoosData^.MinMax[i].T_Min := 100;
                  DoosData^.MinMax[i].U_Max := 300;
                  DoosData^.MinMax[i].U_Min := 30;
                  DoosData^.MinMax[i].V_Max := 300;
                  DoosData^.MinMax[i].V_Min := 30;
                  DoosData^.MinMax[i].W_Max := 1280;
                  DoosData^.MinMax[i].W_Min := 0;
                  DoosData^.MinMax[i].X_Max := 300;
                  DoosData^.MinMax[i].X_Min := 30;
                  DoosData^.MinMax[i].Y_Max := 980;
                  DoosData^.MinMax[i].Y_Min := 155;
                  DoosData^.MinMax[i].Z_Max := 3000;
                  DoosData^.MinMax[i].Z_Min := 0;
                  DoosData^.MinMax[i].Offset_Max := 725;
                  DoosData^.MinMax[i].Offset_Min := 0;

            //6-punt in/in 1450
            elsif i = 10 then

                  DoosData^.MinMax[i].T_Max := 2000;
                  DoosData^.MinMax[i].T_Min := 100;
                  DoosData^.MinMax[i].U_Max := 300;
                  DoosData^.MinMax[i].U_Min := 30;
                  DoosData^.MinMax[i].V_Max := 300;
                  DoosData^.MinMax[i].V_Min := 30;
                  DoosData^.MinMax[i].W_Max := 1280;
                  DoosData^.MinMax[i].W_Min := 0;
                  DoosData^.MinMax[i].X_Max := 300;
                  DoosData^.MinMax[i].X_Min := 30;
                  DoosData^.MinMax[i].Y_Max := 980;
                  DoosData^.MinMax[i].Y_Min := 155;
                  DoosData^.MinMax[i].Z_Max := 3000;
                  DoosData^.MinMax[i].Z_Min := 0;
                  DoosData^.MinMax[i].Offset_Max := 725;
                  DoosData^.MinMax[i].Offset_Min := 0;

            //3-punt (gespiegeld) 1450
            elsif i = 11 then

                  DoosData^.MinMax[i].T_Max := 2000;
                  DoosData^.MinMax[i].T_Min := 100;
                  DoosData^.MinMax[i].U_Max := 250;
                  DoosData^.MinMax[i].U_Min := 40;
                  DoosData^.MinMax[i].V_Max := 250;
                  DoosData^.MinMax[i].V_Min := 40;
                  DoosData^.MinMax[i].W_Max := 1450;
                  DoosData^.MinMax[i].W_Min := 320;
                  DoosData^.MinMax[i].X_Max := 525;
                  DoosData^.MinMax[i].X_Min := 50;
                  DoosData^.MinMax[i].Y_Max := 525;
                  DoosData^.MinMax[i].Y_Min := 75;
                  DoosData^.MinMax[i].Z_Max := 3000;
                  DoosData^.MinMax[i].Z_Min := 0;
                  DoosData^.MinMax[i].Offset_Max := 725;
                  DoosData^.MinMax[i].Offset_Min := 0;

            //3-punt (Storaenzo Jonkoping) 1450
            elsif i = 12 then

                  DoosData^.MinMax[i].T_Max := 2000;
                  DoosData^.MinMax[i].T_Min := 100;
                  DoosData^.MinMax[i].U_Max := 250;
                  DoosData^.MinMax[i].U_Min := 40;
                  DoosData^.MinMax[i].V_Max := 250;
                  DoosData^.MinMax[i].V_Min := 40;
                  DoosData^.MinMax[i].W_Max := 1450;
                  DoosData^.MinMax[i].W_Min := 320;
                  DoosData^.MinMax[i].X_Max := 525;
                  DoosData^.MinMax[i].X_Min := 50;
                  DoosData^.MinMax[i].Y_Max := 525;
                  DoosData^.MinMax[i].Y_Min := 75;
                  DoosData^.MinMax[i].Z_Max := 3000;
                  DoosData^.MinMax[i].Z_Min := 0;
                  DoosData^.MinMax[i].Offset_Max := 725;
                  DoosData^.MinMax[i].Offset_Min := 0;

           //langsnaad2 1450
            elsif i = 13 then

                  DoosData^.MinMax[i].T_Max := 2000;
                  DoosData^.MinMax[i].T_Min := 100;
                  DoosData^.MinMax[i].U_Max := 300;
                  DoosData^.MinMax[i].U_Min := 40;
                  DoosData^.MinMax[i].V_Max := 300;
                  DoosData^.MinMax[i].V_Min := 40;
                  DoosData^.MinMax[i].W_Max := 1450;
                  DoosData^.MinMax[i].W_Min := 320;
                  DoosData^.MinMax[i].X_Max := 525;
                  DoosData^.MinMax[i].X_Min := 40;
                  DoosData^.MinMax[i].Y_Max := 525;
                  DoosData^.MinMax[i].Y_Min := 75;
                  DoosData^.MinMax[i].Z_Max := 3000;
                  DoosData^.MinMax[i].Z_Min := 0;
                  DoosData^.MinMax[i].Offset_Max := 725;
                  DoosData^.MinMax[i].Offset_Min := 0;

            //3-punt2 1450
            elsif i = 14 then

                  DoosData^.MinMax[i].T_Max := 2000;
                  DoosData^.MinMax[i].T_Min := 100;
                  DoosData^.MinMax[i].U_Max := 250;
                  DoosData^.MinMax[i].U_Min := 40;
                  DoosData^.MinMax[i].V_Max := 250;
                  DoosData^.MinMax[i].V_Min := 40;
                  DoosData^.MinMax[i].W_Max := 1450;
                  DoosData^.MinMax[i].W_Min := 320;
                  DoosData^.MinMax[i].X_Max := 525;
                  DoosData^.MinMax[i].X_Min := 50;
                  DoosData^.MinMax[i].Y_Max := 525;
                  DoosData^.MinMax[i].Y_Min := 75;
                  DoosData^.MinMax[i].Z_Max := 3000;
                  DoosData^.MinMax[i].Z_Min := 0;
                  DoosData^.MinMax[i].Offset_Max := 725;
                  DoosData^.MinMax[i].Offset_Min := 0;

           end_if;
        end_for;
  end_if;

  if    Presets_MinMax =  m1700 then

        for i:= 1 to 14 do

            DoosData^.MinMax[i].Max_Invoer_Lengte  := 2000;
            DoosData^.MinMax[i].Max_Invoer_Breedte := 1700;

              //langsnaad 1700
            if    i = 1 then

                  DoosData^.MinMax[i].T_Max := 2000;
                  DoosData^.MinMax[i].T_Min := 160;
                  DoosData^.MinMax[i].U_Max := 300;
                  DoosData^.MinMax[i].U_Min := 40;
                  DoosData^.MinMax[i].V_Max := 0;
                  DoosData^.MinMax[i].V_Min := 0;
                  DoosData^.MinMax[i].W_Max := 1700;
                  DoosData^.MinMax[i].W_Min := 380;
                  DoosData^.MinMax[i].X_Max := 540;
                  DoosData^.MinMax[i].X_Min := 40;
                  DoosData^.MinMax[i].Y_Max := 640;
                  DoosData^.MinMax[i].Y_Min := 90;
                  DoosData^.MinMax[i].Z_Max := 3000;
                  DoosData^.MinMax[i].Z_Min := 0;
                  DoosData^.MinMax[i].Offset_Max := 850;
                  DoosData^.MinMax[i].Offset_Min := 0;

            //3-punt 1700
            elsif i = 2 then

                  DoosData^.MinMax[i].T_Max := 2000;
                  DoosData^.MinMax[i].T_Min := 160;
                  DoosData^.MinMax[i].U_Max := 250;
                  DoosData^.MinMax[i].U_Min := 40;
                  DoosData^.MinMax[i].V_Max := 250;
                  DoosData^.MinMax[i].V_Min := 40;
                  DoosData^.MinMax[i].W_Max := 1700;
                  DoosData^.MinMax[i].W_Min := 380;
                  DoosData^.MinMax[i].X_Max := 640;
                  DoosData^.MinMax[i].X_Min := 50;
                  DoosData^.MinMax[i].Y_Max := 640;
                  DoosData^.MinMax[i].Y_Min := 90;
                  DoosData^.MinMax[i].Z_Max := 3000;
                  DoosData^.MinMax[i].Z_Min := 0;
                  DoosData^.MinMax[i].Offset_Max := 850;
                  DoosData^.MinMax[i].Offset_Min := 0;

            //3-punt vakverdeling 1700
            elsif i = 3 then

                  DoosData^.MinMax[i].T_Max := 2000;
                  DoosData^.MinMax[i].T_Min := 320;
                  DoosData^.MinMax[i].U_Max := 300;
                  DoosData^.MinMax[i].U_Min := 30;
                  DoosData^.MinMax[i].V_Max := 300;
                  DoosData^.MinMax[i].V_Min := 30;
                  DoosData^.MinMax[i].W_Max := 1500;
                  DoosData^.MinMax[i].W_Min := 400;
                  DoosData^.MinMax[i].X_Max := 640;
                  DoosData^.MinMax[i].X_Min := 110;
                  DoosData^.MinMax[i].Y_Max := 640;
                  DoosData^.MinMax[i].Y_Min := 90;
                  DoosData^.MinMax[i].Z_Max := 3000;
                  DoosData^.MinMax[i].Z_Min := 0;
                  DoosData^.MinMax[i].Offset_Max := 850;
                  DoosData^.MinMax[i].Offset_Min := 0;

            //4-punt infold 1700
            elsif i = 4 then

                  DoosData^.MinMax[i].T_Max := 2000;
                  DoosData^.MinMax[i].T_Min := 150;
                  DoosData^.MinMax[i].U_Max := 300;
                  DoosData^.MinMax[i].U_Min := 30;
                  DoosData^.MinMax[i].V_Max := 300;
                  DoosData^.MinMax[i].V_Min := 30;
                  DoosData^.MinMax[i].W_Max := 0;
                  DoosData^.MinMax[i].W_Min := 0;
                  DoosData^.MinMax[i].X_Max := 300;
                  DoosData^.MinMax[i].X_Min := 30;
                  DoosData^.MinMax[i].Y_Max := 1180;
                  DoosData^.MinMax[i].Y_Min := 185;
                  DoosData^.MinMax[i].Z_Max := 3000;
                  DoosData^.MinMax[i].Z_Min := 0;
                  DoosData^.MinMax[i].Offset_Max := 850;
                  DoosData^.MinMax[i].Offset_Min := 0;

            //4-punt outfold 1700
            elsif i = 5 then

                  DoosData^.MinMax[i].T_Max := 2000;
                  DoosData^.MinMax[i].T_Min := 150;
                  DoosData^.MinMax[i].U_Max := 300;
                  DoosData^.MinMax[i].U_Min := 30;
                  DoosData^.MinMax[i].V_Max := 300;
                  DoosData^.MinMax[i].V_Min := 30;
                  DoosData^.MinMax[i].W_Max := 0;
                  DoosData^.MinMax[i].W_Min := 0;
                  DoosData^.MinMax[i].X_Max := 300;
                  DoosData^.MinMax[i].X_Min := 30;
                  DoosData^.MinMax[i].Y_Max := 1180;
                  DoosData^.MinMax[i].Y_Min := 185;
                  DoosData^.MinMax[i].Z_Max := 3000;
                  DoosData^.MinMax[i].Z_Min := 0;
                  DoosData^.MinMax[i].Offset_Max := 850;
                  DoosData^.MinMax[i].Offset_Min := 0;

            //4-punt met deksel 1700
            elsif i = 6 then

                  DoosData^.MinMax[i].T_Max := 2000;
                  DoosData^.MinMax[i].T_Min := 150;
                  DoosData^.MinMax[i].U_Max := 300;
                  DoosData^.MinMax[i].U_Min := 30;
                  DoosData^.MinMax[i].V_Max := 300;
                  DoosData^.MinMax[i].V_Min := 30;
                  DoosData^.MinMax[i].W_Max := 1580;
                  DoosData^.MinMax[i].W_Min := 0;
                  DoosData^.MinMax[i].X_Max := 300;
                  DoosData^.MinMax[i].X_Min := 30;
                  DoosData^.MinMax[i].Y_Max := 1180;
                  DoosData^.MinMax[i].Y_Min := 185;
                  DoosData^.MinMax[i].Z_Max := 3000;
                  DoosData^.MinMax[i].Z_Min := 0;
                  DoosData^.MinMax[i].Offset_Max := 850;
                  DoosData^.MinMax[i].Offset_Min := 0;

            //4-punt dubbele wand 1700
            elsif i = 7 then

                  DoosData^.MinMax[i].T_Max := 2000;
                  DoosData^.MinMax[i].T_Min := 150;
                  DoosData^.MinMax[i].U_Max := 300;
                  DoosData^.MinMax[i].U_Min := 30;
                  DoosData^.MinMax[i].V_Max := 300;
                  DoosData^.MinMax[i].V_Min := 30;
                  DoosData^.MinMax[i].W_Max := 1580;
                  DoosData^.MinMax[i].W_Min := 0;
                  DoosData^.MinMax[i].X_Max := 300;
                  DoosData^.MinMax[i].X_Min := 30;
                  DoosData^.MinMax[i].Y_Max := 1180;
                  DoosData^.MinMax[i].Y_Min := 185;
                  DoosData^.MinMax[i].Z_Max := 3000;
                  DoosData^.MinMax[i].Z_Min := 0;
                  DoosData^.MinMax[i].Offset_Max := 850;
                  DoosData^.MinMax[i].Offset_Min := 0;

            //6-punt in/in 1700
            elsif i = 8 then

                  DoosData^.MinMax[i].T_Max := 2000;
                  DoosData^.MinMax[i].T_Min := 150;
                  DoosData^.MinMax[i].U_Max := 300;
                  DoosData^.MinMax[i].U_Min := 30;
                  DoosData^.MinMax[i].V_Max := 300;
                  DoosData^.MinMax[i].V_Min := 30;
                  DoosData^.MinMax[i].W_Max := 1580;
                  DoosData^.MinMax[i].W_Min := 0;
                  DoosData^.MinMax[i].X_Max := 300;
                  DoosData^.MinMax[i].X_Min := 30;
                  DoosData^.MinMax[i].Y_Max := 1180;
                  DoosData^.MinMax[i].Y_Min := 185;
                  DoosData^.MinMax[i].Z_Max := 3000;
                  DoosData^.MinMax[i].Z_Min := 0;
                  DoosData^.MinMax[i].Offset_Max := 850;
                  DoosData^.MinMax[i].Offset_Min := 0;

            //6-punt in/out 1700
            elsif i = 9 then

                  DoosData^.MinMax[i].T_Max := 2000;
                  DoosData^.MinMax[i].T_Min := 150;
                  DoosData^.MinMax[i].U_Max := 300;
                  DoosData^.MinMax[i].U_Min := 30;
                  DoosData^.MinMax[i].V_Max := 300;
                  DoosData^.MinMax[i].V_Min := 30;
                  DoosData^.MinMax[i].W_Max := 1580;
                  DoosData^.MinMax[i].W_Min := 0;
                  DoosData^.MinMax[i].X_Max := 300;
                  DoosData^.MinMax[i].X_Min := 30;
                  DoosData^.MinMax[i].Y_Max := 1180;
                  DoosData^.MinMax[i].Y_Min := 185;
                  DoosData^.MinMax[i].Z_Max := 3000;
                  DoosData^.MinMax[i].Z_Min := 0;
                  DoosData^.MinMax[i].Offset_Max := 850;
                  DoosData^.MinMax[i].Offset_Min := 0;

            //6-punt in/in 1700
            elsif i = 10 then

                  DoosData^.MinMax[i].T_Max := 2000;
                  DoosData^.MinMax[i].T_Min := 150;
                  DoosData^.MinMax[i].U_Max := 300;
                  DoosData^.MinMax[i].U_Min := 30;
                  DoosData^.MinMax[i].V_Max := 300;
                  DoosData^.MinMax[i].V_Min := 30;
                  DoosData^.MinMax[i].W_Max := 1580;
                  DoosData^.MinMax[i].W_Min := 0;
                  DoosData^.MinMax[i].X_Max := 300;
                  DoosData^.MinMax[i].X_Min := 30;
                  DoosData^.MinMax[i].Y_Max := 1180;
                  DoosData^.MinMax[i].Y_Min := 185;
                  DoosData^.MinMax[i].Z_Max := 3000;
                  DoosData^.MinMax[i].Z_Min := 0;
                  DoosData^.MinMax[i].Offset_Max := 850;
                  DoosData^.MinMax[i].Offset_Min := 0;

            //3-punt (gespiegeld) 1700
            elsif i = 11 then

                  DoosData^.MinMax[i].T_Max := 2000;
                  DoosData^.MinMax[i].T_Min := 160;
                  DoosData^.MinMax[i].U_Max := 250;
                  DoosData^.MinMax[i].U_Min := 40;
                  DoosData^.MinMax[i].V_Max := 250;
                  DoosData^.MinMax[i].V_Min := 40;
                  DoosData^.MinMax[i].W_Max := 1700;
                  DoosData^.MinMax[i].W_Min := 380;
                  DoosData^.MinMax[i].X_Max := 640;
                  DoosData^.MinMax[i].X_Min := 50;
                  DoosData^.MinMax[i].Y_Max := 640;
                  DoosData^.MinMax[i].Y_Min := 90;
                  DoosData^.MinMax[i].Z_Max := 300;
                  DoosData^.MinMax[i].Z_Min := 0;
                  DoosData^.MinMax[i].Offset_Max := 850;
                  DoosData^.MinMax[i].Offset_Min := 0;

            //3-punt (Storaenzo Jonkoping) 1700
            elsif i = 12 then

                  DoosData^.MinMax[i].T_Max := 2000;
                  DoosData^.MinMax[i].T_Min := 160;
                  DoosData^.MinMax[i].U_Max := 250;
                  DoosData^.MinMax[i].U_Min := 40;
                  DoosData^.MinMax[i].V_Max := 250;
                  DoosData^.MinMax[i].V_Min := 40;
                  DoosData^.MinMax[i].W_Max := 1700;
                  DoosData^.MinMax[i].W_Min := 380;
                  DoosData^.MinMax[i].X_Max := 640;
                  DoosData^.MinMax[i].X_Min := 50;
                  DoosData^.MinMax[i].Y_Max := 640;
                  DoosData^.MinMax[i].Y_Min := 90;
                  DoosData^.MinMax[i].Z_Max := 300;
                  DoosData^.MinMax[i].Z_Min := 0;
                  DoosData^.MinMax[i].Offset_Max := 850;
                  DoosData^.MinMax[i].Offset_Min := 0;

            //langsnaad2 1700
            elsif i = 13 then

                  DoosData^.MinMax[i].T_Max := 2000;
                  DoosData^.MinMax[i].T_Min := 160;
                  DoosData^.MinMax[i].U_Max := 300;
                  DoosData^.MinMax[i].U_Min := 40;
                  DoosData^.MinMax[i].V_Max := 300;
                  DoosData^.MinMax[i].V_Min := 40;
                  DoosData^.MinMax[i].W_Max := 1700;
                  DoosData^.MinMax[i].W_Min := 380;
                  DoosData^.MinMax[i].X_Max := 540;
                  DoosData^.MinMax[i].X_Min := 40;
                  DoosData^.MinMax[i].Y_Max := 640;
                  DoosData^.MinMax[i].Y_Min := 90;
                  DoosData^.MinMax[i].Z_Max := 300;
                  DoosData^.MinMax[i].Z_Min := 0;
                  DoosData^.MinMax[i].Offset_Max := 850;
                  DoosData^.MinMax[i].Offset_Min := 0;

            //3-punt2 1700
            elsif i = 14 then

                  DoosData^.MinMax[i].T_Max := 2000;
                  DoosData^.MinMax[i].T_Min := 160;
                  DoosData^.MinMax[i].U_Max := 250;
                  DoosData^.MinMax[i].U_Min := 40;
                  DoosData^.MinMax[i].V_Max := 250;
                  DoosData^.MinMax[i].V_Min := 40;
                  DoosData^.MinMax[i].W_Max := 1700;
                  DoosData^.MinMax[i].W_Min := 380;
                  DoosData^.MinMax[i].X_Max := 640;
                  DoosData^.MinMax[i].X_Min := 50;
                  DoosData^.MinMax[i].Y_Max := 640;
                  DoosData^.MinMax[i].Y_Min := 90;
                  DoosData^.MinMax[i].Z_Max := 300;
                  DoosData^.MinMax[i].Z_Min := 0;
                  DoosData^.MinMax[i].Offset_Max := 850;
                  DoosData^.MinMax[i].Offset_Min := 0;
            end_if;
        end_for;
  end_if;

  if    Presets_MinMax =  m1900 then

        for i:= 1 to 14 do

            DoosData^.MinMax[i].Max_Invoer_Lengte  := 2000;
            DoosData^.MinMax[i].Max_Invoer_Breedte := 1900;

              //langsnaad 1900
            if    i = 1 then

                  DoosData^.MinMax[i].T_Max := 2000;
                  DoosData^.MinMax[i].T_Min := 160;
                  DoosData^.MinMax[i].U_Max := 300;
                  DoosData^.MinMax[i].U_Min := 50;
                  DoosData^.MinMax[i].V_Max := 0;
                  DoosData^.MinMax[i].V_Min := 0;
                  DoosData^.MinMax[i].W_Max := 1900;
                  DoosData^.MinMax[i].W_Min := 510;
                  DoosData^.MinMax[i].X_Max := 740;
                  DoosData^.MinMax[i].X_Min := 50;
                  DoosData^.MinMax[i].Y_Max := 740;
                  DoosData^.MinMax[i].Y_Min := 150;
                  DoosData^.MinMax[i].Z_Max := 300;
                  DoosData^.MinMax[i].Z_Min := 0;
                  DoosData^.MinMax[i].Offset_Max := 950;
                  DoosData^.MinMax[i].Offset_Min := 0;

            //3-punt 1900
            elsif i = 2 then

                  DoosData^.MinMax[i].T_Max := 2000;
                  DoosData^.MinMax[i].T_Min := 160;
                  DoosData^.MinMax[i].U_Max := 300;
                  DoosData^.MinMax[i].U_Min := 50;
                  DoosData^.MinMax[i].V_Max := 300;
                  DoosData^.MinMax[i].V_Min := 50;
                  DoosData^.MinMax[i].W_Max := 1900;
                  DoosData^.MinMax[i].W_Min := 510;
                  DoosData^.MinMax[i].X_Max := 740;
                  DoosData^.MinMax[i].X_Min := 50;
                  DoosData^.MinMax[i].Y_Max := 740;
                  DoosData^.MinMax[i].Y_Min := 150;
                  DoosData^.MinMax[i].Z_Max := 300;
                  DoosData^.MinMax[i].Z_Min := 0;
                  DoosData^.MinMax[i].Offset_Max := 950;
                  DoosData^.MinMax[i].Offset_Min := 0;

            //3-punt vakverdeling 1900
            elsif i = 3 then

                  DoosData^.MinMax[i].T_Max := 2000;
                  DoosData^.MinMax[i].T_Min := 320;
                  DoosData^.MinMax[i].U_Max := 300;
                  DoosData^.MinMax[i].U_Min := 30;
                  DoosData^.MinMax[i].V_Max := 300;
                  DoosData^.MinMax[i].V_Min := 30;
                  DoosData^.MinMax[i].W_Max := 1700;
                  DoosData^.MinMax[i].W_Min := 500;
                  DoosData^.MinMax[i].X_Max := 740;
                  DoosData^.MinMax[i].X_Min := 150;
                  DoosData^.MinMax[i].Y_Max := 740;
                  DoosData^.MinMax[i].Y_Min := 100;
                  DoosData^.MinMax[i].Z_Max := 300;
                  DoosData^.MinMax[i].Z_Min := 0;
                  DoosData^.MinMax[i].Offset_Max := 950;
                  DoosData^.MinMax[i].Offset_Min := 0;

            //4-punt infold 1900
            elsif i = 4 then

                  DoosData^.MinMax[i].T_Max := 2000;
                  DoosData^.MinMax[i].T_Min := 150;
                  DoosData^.MinMax[i].U_Max := 300;
                  DoosData^.MinMax[i].U_Min := 30;
                  DoosData^.MinMax[i].V_Max := 300;
                  DoosData^.MinMax[i].V_Min := 30;
                  DoosData^.MinMax[i].W_Max := 0;
                  DoosData^.MinMax[i].W_Min := 0;
                  DoosData^.MinMax[i].X_Max := 300;
                  DoosData^.MinMax[i].X_Min := 30;
                  DoosData^.MinMax[i].Y_Max := 1180;
                  DoosData^.MinMax[i].Y_Min := 250;
                  DoosData^.MinMax[i].Z_Max := 300;
                  DoosData^.MinMax[i].Z_Min := 0;
                  DoosData^.MinMax[i].Offset_Max := 950;
                  DoosData^.MinMax[i].Offset_Min := 0;

            //4-punt outfold 1900
            elsif i = 5 then

                  DoosData^.MinMax[i].T_Max := 2000;
                  DoosData^.MinMax[i].T_Min := 150;
                  DoosData^.MinMax[i].U_Max := 300;
                  DoosData^.MinMax[i].U_Min := 30;
                  DoosData^.MinMax[i].V_Max := 300;
                  DoosData^.MinMax[i].V_Min := 30;
                  DoosData^.MinMax[i].W_Max := 0;
                  DoosData^.MinMax[i].W_Min := 0;
                  DoosData^.MinMax[i].X_Max := 300;
                  DoosData^.MinMax[i].X_Min := 30;
                  DoosData^.MinMax[i].Y_Max := 1180;
                  DoosData^.MinMax[i].Y_Min := 250;
                  DoosData^.MinMax[i].Z_Max := 300;
                  DoosData^.MinMax[i].Z_Min := 0;
                  DoosData^.MinMax[i].Offset_Max := 950;
                  DoosData^.MinMax[i].Offset_Min := 0;

            //4-punt met deksel 1900
            elsif i = 6 then

                  DoosData^.MinMax[i].T_Max := 2000;
                  DoosData^.MinMax[i].T_Min := 150;
                  DoosData^.MinMax[i].U_Max := 300;
                  DoosData^.MinMax[i].U_Min := 30;
                  DoosData^.MinMax[i].V_Max := 300;
                  DoosData^.MinMax[i].V_Min := 30;
                  DoosData^.MinMax[i].W_Max := 1770;
                  DoosData^.MinMax[i].W_Min := 0;
                  DoosData^.MinMax[i].X_Max := 300;
                  DoosData^.MinMax[i].X_Min := 30;
                  DoosData^.MinMax[i].Y_Max := 1180;
                  DoosData^.MinMax[i].Y_Min := 250;
                  DoosData^.MinMax[i].Z_Max := 300;
                  DoosData^.MinMax[i].Z_Min := 0;
                  DoosData^.MinMax[i].Offset_Max := 950;
                  DoosData^.MinMax[i].Offset_Min := 0;

            //4-punt dubbele wand 1900
            elsif i = 7 then

                  DoosData^.MinMax[i].T_Max := 2000;
                  DoosData^.MinMax[i].T_Min := 150;
                  DoosData^.MinMax[i].U_Max := 300;
                  DoosData^.MinMax[i].U_Min := 30;
                  DoosData^.MinMax[i].V_Max := 300;
                  DoosData^.MinMax[i].V_Min := 30;
                  DoosData^.MinMax[i].W_Max := 1770;
                  DoosData^.MinMax[i].W_Min := 0;
                  DoosData^.MinMax[i].X_Max := 300;
                  DoosData^.MinMax[i].X_Min := 30;
                  DoosData^.MinMax[i].Y_Max := 1180;
                  DoosData^.MinMax[i].Y_Min := 250;
                  DoosData^.MinMax[i].Z_Max := 300;
                  DoosData^.MinMax[i].Z_Min := 0;
                  DoosData^.MinMax[i].Offset_Max := 950;
                  DoosData^.MinMax[i].Offset_Min := 0;

            //6-punt in/in 1900
            elsif i = 8 then

                  DoosData^.MinMax[i].T_Max := 2000;
                  DoosData^.MinMax[i].T_Min := 150;
                  DoosData^.MinMax[i].U_Max := 300;
                  DoosData^.MinMax[i].U_Min := 30;
                  DoosData^.MinMax[i].V_Max := 300;
                  DoosData^.MinMax[i].V_Min := 30;
                  DoosData^.MinMax[i].W_Max := 1770;
                  DoosData^.MinMax[i].W_Min := 0;
                  DoosData^.MinMax[i].X_Max := 300;
                  DoosData^.MinMax[i].X_Min := 30;
                  DoosData^.MinMax[i].Y_Max := 1180;
                  DoosData^.MinMax[i].Y_Min := 250;
                  DoosData^.MinMax[i].Z_Max := 300;
                  DoosData^.MinMax[i].Z_Min := 0;
                  DoosData^.MinMax[i].Offset_Max := 950;
                  DoosData^.MinMax[i].Offset_Min := 0;

            //6-punt in/out 1900
            elsif i = 9 then

                  DoosData^.MinMax[i].T_Max := 2000;
                  DoosData^.MinMax[i].T_Min := 150;
                  DoosData^.MinMax[i].U_Max := 300;
                  DoosData^.MinMax[i].U_Min := 30;
                  DoosData^.MinMax[i].V_Max := 300;
                  DoosData^.MinMax[i].V_Min := 30;
                  DoosData^.MinMax[i].W_Max := 1770;
                  DoosData^.MinMax[i].W_Min := 0;
                  DoosData^.MinMax[i].X_Max := 300;
                  DoosData^.MinMax[i].X_Min := 30;
                  DoosData^.MinMax[i].Y_Max := 1180;
                  DoosData^.MinMax[i].Y_Min := 250;
                  DoosData^.MinMax[i].Z_Max := 300;
                  DoosData^.MinMax[i].Z_Min := 0;
                  DoosData^.MinMax[i].Offset_Max := 950;
                  DoosData^.MinMax[i].Offset_Min := 0;

            //6-punt in/in 1900
            elsif i = 10 then

                  DoosData^.MinMax[i].T_Max := 2000;
                  DoosData^.MinMax[i].T_Min := 150;
                  DoosData^.MinMax[i].U_Max := 300;
                  DoosData^.MinMax[i].U_Min := 30;
                  DoosData^.MinMax[i].V_Max := 300;
                  DoosData^.MinMax[i].V_Min := 30;
                  DoosData^.MinMax[i].W_Max := 1770;
                  DoosData^.MinMax[i].W_Min := 0;
                  DoosData^.MinMax[i].X_Max := 300;
                  DoosData^.MinMax[i].X_Min := 30;
                  DoosData^.MinMax[i].Y_Max := 1180;
                  DoosData^.MinMax[i].Y_Min := 250;
                  DoosData^.MinMax[i].Z_Max := 300;
                  DoosData^.MinMax[i].Z_Min := 0;
                  DoosData^.MinMax[i].Offset_Max := 950;
                  DoosData^.MinMax[i].Offset_Min := 0;

            //3-punt (gespiegeld) 1900
            elsif i = 11 then

                  DoosData^.MinMax[i].T_Max := 2000;
                  DoosData^.MinMax[i].T_Min := 160;
                  DoosData^.MinMax[i].U_Max := 300;
                  DoosData^.MinMax[i].U_Min := 50;
                  DoosData^.MinMax[i].V_Max := 300;
                  DoosData^.MinMax[i].V_Min := 50;
                  DoosData^.MinMax[i].W_Max := 1900;
                  DoosData^.MinMax[i].W_Min := 510;
                  DoosData^.MinMax[i].X_Max := 740;
                  DoosData^.MinMax[i].X_Min := 50;
                  DoosData^.MinMax[i].Y_Max := 740;
                  DoosData^.MinMax[i].Y_Min := 150;
                  DoosData^.MinMax[i].Z_Max := 300;
                  DoosData^.MinMax[i].Z_Min := 0;
                  DoosData^.MinMax[i].Offset_Max := 950;
                  DoosData^.MinMax[i].Offset_Min := 0;

            //3-punt (Storaenzo Jonkoping) 1900
            elsif i = 12 then

                  DoosData^.MinMax[i].T_Max := 2000;
                  DoosData^.MinMax[i].T_Min := 160;
                  DoosData^.MinMax[i].U_Max := 300;
                  DoosData^.MinMax[i].U_Min := 50;
                  DoosData^.MinMax[i].V_Max := 300;
                  DoosData^.MinMax[i].V_Min := 50;
                  DoosData^.MinMax[i].W_Max := 1900;
                  DoosData^.MinMax[i].W_Min := 510;
                  DoosData^.MinMax[i].X_Max := 740;
                  DoosData^.MinMax[i].X_Min := 50;
                  DoosData^.MinMax[i].Y_Max := 740;
                  DoosData^.MinMax[i].Y_Min := 150;
                  DoosData^.MinMax[i].Z_Max := 300;
                  DoosData^.MinMax[i].Z_Min := 0;
                  DoosData^.MinMax[i].Offset_Max := 950;
                  DoosData^.MinMax[i].Offset_Min := 0;

            //langsnaad2 1900
            elsif i = 13 then

                  DoosData^.MinMax[i].T_Max := 2000;
                  DoosData^.MinMax[i].T_Min := 160;
                  DoosData^.MinMax[i].U_Max := 300;
                  DoosData^.MinMax[i].U_Min := 50;
                  DoosData^.MinMax[i].V_Max := 300;
                  DoosData^.MinMax[i].V_Min := 50;
                  DoosData^.MinMax[i].W_Max := 1900;
                  DoosData^.MinMax[i].W_Min := 510;
                  DoosData^.MinMax[i].X_Max := 740;
                  DoosData^.MinMax[i].X_Min := 50;
                  DoosData^.MinMax[i].Y_Max := 740;
                  DoosData^.MinMax[i].Y_Min := 150;
                  DoosData^.MinMax[i].Z_Max := 300;
                  DoosData^.MinMax[i].Z_Min := 0;
                  DoosData^.MinMax[i].Offset_Max := 950;
                  DoosData^.MinMax[i].Offset_Min := 0;

            //3-punt2 1900
            elsif i = 14 then

                  DoosData^.MinMax[i].T_Max := 2000;
                  DoosData^.MinMax[i].T_Min := 160;
                  DoosData^.MinMax[i].U_Max := 300;
                  DoosData^.MinMax[i].U_Min := 50;
                  DoosData^.MinMax[i].V_Max := 300;
                  DoosData^.MinMax[i].V_Min := 50;
                  DoosData^.MinMax[i].W_Max := 1900;
                  DoosData^.MinMax[i].W_Min := 510;
                  DoosData^.MinMax[i].X_Max := 740;
                  DoosData^.MinMax[i].X_Min := 50;
                  DoosData^.MinMax[i].Y_Max := 740;
                  DoosData^.MinMax[i].Y_Min := 150;
                  DoosData^.MinMax[i].Z_Max := 300;
                  DoosData^.MinMax[i].Z_Min := 0;
                  DoosData^.MinMax[i].Offset_Max := 950;
                  DoosData^.MinMax[i].Offset_Min := 0;
           end_if;
        end_for;
  end_if;

  if    Presets_MinMax =  m2300 then

        for i:= 1 to 14 do

            DoosData^.MinMax[i].Max_Invoer_Lengte  := 2000;
            DoosData^.MinMax[i].Max_Invoer_Breedte := 2300;

              //langsnaad 2300
            if    i = 1 then

                  DoosData^.MinMax[i].T_Max := 2000;
                  DoosData^.MinMax[i].T_Min := 160;
                  DoosData^.MinMax[i].U_Max := 300;
                  DoosData^.MinMax[i].U_Min := 50;
                  DoosData^.MinMax[i].V_Max := 0;
                  DoosData^.MinMax[i].V_Min := 0;
                  DoosData^.MinMax[i].W_Max := 2300;
                  DoosData^.MinMax[i].W_Min := 510;
                  DoosData^.MinMax[i].X_Max := 820;
                  DoosData^.MinMax[i].X_Min := 50;
                  DoosData^.MinMax[i].Y_Max := 820;
                  DoosData^.MinMax[i].Y_Min := 150;
                  DoosData^.MinMax[i].Z_Max := 300;
                  DoosData^.MinMax[i].Z_Min := 0;
                  DoosData^.MinMax[i].Offset_Max := 1150;
                  DoosData^.MinMax[i].Offset_Min := 0;
